  MoveL 10079 to (-40.2, 152.67, 144.49) mm, rotated rx -180 ry 0 rz 180 deg; joints [-142.671, 73.983, -86.26, 142.029, 80.265, 7.518]
  Call Extruder(400.11411)
  MoveL 10080 to (-40.24, 152.44, 144.49) mm, rotated rx -180 ry 0 rz 180 deg; joints [-142.718, 73.976, -86.267, 142.076, 80.248, 7.518]
  MoveL 10081 to (-40.24, 152.44, 144.49) mm, rotated rx -180 ry 0 rz 180 deg; joints [-142.718, 73.976, -86.267, 142.076, 80.248, 7.518]
  Call Extruder(400.25109)
  MoveL 10082 to (-40.29, 152.2, 144.49) mm, rotated rx 180 ry 0 rz -180 deg; joints [-142.77, 73.969, -86.275, 142.127, 80.23, 7.518]
  MoveL 10083 to (-40.29, 152.2, 144.49) mm, rotated rx 180 ry 0 rz -180 deg; joints [-142.77, 73.969, -86.275, 142.127, 80.23, 7.518]
  Call Extruder(400.38745)
  MoveL 10084 to (-40.34, 151.95, 144.49) mm, rotated rx 180 ry 0 rz -180 deg; joints [-142.822, 73.961, -86.282, 142.177, 80.211, 7.519]
  MoveL 10085 to (-40.34, 151.95, 144.49) mm, rotated rx 180 ry 0 rz -180 deg; joints [-142.822, 73.961, -86.282, 142.177, 80.211, 7.519]
  Call Extruder(400.52321)
  MoveL 10086 to (-40.39, 151.7, 144.49) mm, rotated rx -180 ry 0 rz -180 deg; joints [-142.874, 73.954, -86.29, 142.228, 80.193, 7.519]
  MoveL 10087 to (-40.39, 151.7, 144.49) mm, rotated rx -180 ry 0 rz -180 deg; joints [-142.874, 73.954, -86.29, 142.228, 80.193, 7.519]
  Call Extruder(400.65835)
  MoveL 10088 to (-40.44, 151.45, 144.49) mm, rotated rx -180 ry 0 rz 180 deg; joints [-142.926, 73.947, -86.297, 142.279, 80.174, 7.519]
  MoveL 10089 to (-40.44, 151.45, 144.49) mm, rotated rx -180 ry 0 rz 180 deg; joints [-142.926, 73.947, -86.297, 142.279, 80.174, 7.519]
  Call Extruder(400.79289)
  MoveL 10090 to (-40.49, 151.2, 144.49) mm, rotated rx -180 ry 0 rz 180 deg; joints [-142.978, 73.939, -86.304, 142.33, 80.156, 7.52]
  MoveL 10091 to (-40.49, 151.2, 144.49) mm, rotated rx -180 ry 0 rz 180 deg; joints [-142.978, 73.939, -86.304, 142.33, 80.156, 7.52]
  Call Extruder(400.92681)
  MoveL 10092 to (-40.54, 150.95, 144.49) mm, rotated rx -180 ry 0 rz -180 deg; joints [-143.031, 73.932, -86.312, 142.381, 80.137, 7.52]
  MoveL 10093 to (-40.54, 150.95, 144.49) mm, rotated rx -180 ry 0 rz -180 deg; joints [-143.031, 73.932, -86.312, 142.381, 80.137, 7.52]
  Call Extruder(401.07467)
  MoveL 10094 to (-40.59, 150.67, 144.49) mm, rotated rx -180 ry 0 rz 180 deg; joints [-143.088, 73.923, -86.321, 142.437, 80.116, 7.521]
  MoveL 10095 to (-40.59, 150.67, 144.49) mm, rotated rx -180 ry 0 rz 180 deg; joints [-143.088, 73.923, -86.321, 142.437, 80.116, 7.521]
  Call Extruder(401.23639)
  MoveL 10096 to (-40.64, 150.37, 144.49) mm, rotated rx 180 ry 0 rz 180 deg; joints [-143.15, 73.914, -86.33, 142.498, 80.092, 7.522]
  MoveL 10097 to (-40.64, 150.37, 144.49) mm, rotated rx 180 ry 0 rz 180 deg; joints [-143.15, 73.914, -86.33, 142.498, 80.092, 7.522]
  Call Extruder(401.39739)
  MoveL 10098 to (-40.69, 150.06, 144.49) mm, rotated rx -180 ry 0 rz 180 deg; joints [-143.213, 73.904, -86.34, 142.558, 80.069, 7.523]
  MoveL 10099 to (-40.69, 150.06, 144.49) mm, rotated rx -180 ry 0 rz 180 deg; joints [-143.213, 73.904, -86.34, 142.558, 80.069, 7.523]
  Call Extruder(401.55766)
  MoveL 10100 to (-40.74, 149.76, 144.49) mm, rotated rx 180 ry 0 rz 180 deg; joints [-143.276, 73.894, -86.35, 142.619, 80.045, 7.524]
  MoveL 10101 to (-40.74, 149.76, 144.49) mm, rotated rx 180 ry 0 rz 180 deg; joints [-143.276, 73.894, -86.35, 142.619, 80.045, 7.524]
  Call Extruder(401.71721)
  MoveL 10102 to (-40.78, 149.45, 144.49) mm, rotated rx 180 ry 0 rz 180 deg; joints [-143.338, 73.885, -86.359, 142.681, 80.022, 7.525]
  MoveL 10103 to (-40.78, 149.45, 144.49) mm, rotated rx 180 ry 0 rz 180 deg; joints [-143.338, 73.885, -86.359, 142.681, 80.022, 7.525]
  Call Extruder(401.87602)
  MoveL 10104 to (-40.83, 149.14, 144.49) mm, rotated rx -180 ry 0 rz -180 deg; joints [-143.401, 73.875, -86.369, 142.742, 79.998, 7.526]
  MoveL 10105 to (-40.83, 149.14, 144.49) mm, rotated rx -180 ry 0 rz -180 deg; joints [-143.401, 73.875, -86.369, 142.742, 79.998, 7.526]
  Call Extruder(402.05468)
  MoveL 10106 to (-40.88, 148.8, 144.49) mm, rotated rx 180 ry 0 rz 180 deg; joints [-143.471, 73.864, -86.38, 142.81, 79.971, 7.527]
  MoveL 10107 to (-40.88, 148.8, 144.49) mm, rotated rx 180 ry 0 rz 180 deg; joints [-143.471, 73.864, -86.38, 142.81, 79.971, 7.527]
  Call Extruder(402.25313)
  MoveL 10108 to (-40.93, 148.41, 144.49) mm, rotated rx -180 ry 0 rz 180 deg; joints [-143.549, 73.851, -86.393, 142.885, 79.94, 7.53]
  MoveL 10109 to (-40.93, 148.41, 144.49) mm, rotated rx -180 ry 0 rz 180 deg; joints [-143.549, 73.851, -86.393, 142.885, 79.94, 7.53]
  Call Extruder(402.45070)
  MoveL 10110 to (-40.97, 148.02, 144.49) mm, rotated rx 180 ry 0 rz -180 deg; joints [-143.627, 73.838, -86.406, 142.961, 79.909, 7.532]
  MoveL 10111 to (-40.97, 148.02, 144.49) mm, rotated rx 180 ry 0 rz -180 deg; joints [-143.627, 73.838, -86.406, 142.961, 79.909, 7.532]
  Call Extruder(402.64741)
  MoveL 10112 to (-41.02, 147.63, 144.49) mm, rotated rx -180 ry 0 rz 180 deg; joints [-143.705, 73.825, -86.419, 143.037, 79.878, 7.534]
  MoveL 10113 to (-41.02, 147.63, 144.49) mm, rotated rx -180 ry 0 rz 180 deg; joints [-143.705, 73.825, -86.419, 143.037, 79.878, 7.534]
  Call Extruder(402.84324)
  MoveL 10114 to (-41.06, 147.25, 144.49) mm, rotated rx -180 ry 0 rz 180 deg; joints [-143.783, 73.812, -86.432, 143.112, 79.847, 7.536]
  MoveL 10115 to (-41.06, 147.25, 144.49) mm, rotated rx -180 ry 0 rz 180 deg; joints [-143.783, 73.812, -86.432, 143.112, 79.847, 7.536]
  Call Extruder(403.13864)
  MoveL 10116 to (-41.11, 146.66, 144.49) mm, rotated rx 180 ry 0 rz -180 deg; joints [-143.899, 73.791, -86.453, 143.225, 79.799, 7.541]
  MoveL 10117 to (-41.11, 146.66, 144.49) mm, rotated rx 180 ry 0 rz -180 deg; joints [-143.899, 73.791, -86.453, 143.225, 79.799, 7.541]
  Call Extruder(403.43270)
  MoveL 10118 to (-41.16, 146.07, 144.49) mm, rotated rx 180 ry 0 rz 180 deg; joints [-144.015, 73.77, -86.473, 143.337, 79.75, 7.545]
  MoveL 10119 to (-41.16, 146.07, 144.49) mm, rotated rx 180 ry 0 rz 180 deg; joints [-144.015, 73.77, -86.473, 143.337, 79.75, 7.545]
  Call Extruder(403.72544)
  MoveL 10120 to (-41.2, 145.48, 144.49) mm, rotated rx -180 ry 0 rz 180 deg; joints [-144.131, 73.749, -86.494, 143.45, 79.702, 7.549]
  MoveL 10121 to (-41.2, 145.48, 144.49) mm, rotated rx -180 ry 0 rz 180 deg; joints [-144.131, 73.749, -86.494, 143.45, 79.702, 7.549]
  Call Extruder(404.29889)
  MoveL 10122 to (-41.25, 144.32, 144.49) mm, rotated rx 180 ry 0 rz 180 deg; joints [-144.355, 73.705, -86.536, 143.666, 79.603, 7.561]
  MoveL 10123 to (-41.25, 144.32, 144.49) mm, rotated rx 180 ry 0 rz 180 deg; joints [-144.355, 73.705, -86.536, 143.666, 79.603, 7.561]
  Call Extruder(405.01285)
  MoveL 10124 to (-41.29, 142.86, 144.49) mm, rotated rx 180 ry 0 rz -180 deg; joints [-144.635, 73.65, -86.59, 143.937, 79.478, 7.575]
  Call Extruder(447.07768)
  MoveL 10125 to (-41.29, 57.14, 144.49) mm, rotated rx 180 ry 0 rz -180 deg; joints [-164.153, 70.836, -88.802, 163.384, 72.739, 5.06]
  Call Extruder(447.50624)
  MoveL 10126 to (-41.27, 56.26, 144.49) mm, rotated rx -180 ry 0 rz -180 deg; joints [-164.382, 70.815, -88.815, 163.62, 72.687, 4.999]
  MoveL 10127 to (-41.27, 56.26, 144.49) mm, rotated rx -180 ry 0 rz -180 deg; joints [-164.382, 70.815, -88.815, 163.62, 72.687, 4.999]
  Call Extruder(448.07969)
  MoveL 10128 to (-41.23, 55.1, 144.49) mm, rotated rx -180 ry 0 rz 180 deg; joints [-164.686, 70.787, -88.833, 163.934, 72.615, 4.918]
  MoveL 10129 to (-41.23, 55.1, 144.49) mm, rotated rx -180 ry 0 rz 180 deg; joints [-164.686, 70.787, -88.833, 163.934, 72.615, 4.918]
  Call Extruder(448.51400)
  MoveL 10130 to (-41.18, 54.23, 144.49) mm, rotated rx -180 ry 0 rz 180 deg; joints [-164.915, 70.764, -88.847, 164.17, 72.561, 4.857]
  MoveL 10131 to (-41.18, 54.23, 144.49) mm, rotated rx -180 ry 0 rz 180 deg; joints [-164.915, 70.764, -88.847, 164.17, 72.561, 4.857]
  Call Extruder(448.80807)
  MoveL 10132 to (-41.13, 53.64, 144.49) mm, rotated rx 180 ry 0 rz -180 deg; joints [-165.068, 70.748, -88.857, 164.328, 72.522, 4.817]
  MoveL 10133 to (-41.13, 53.64, 144.49) mm, rotated rx 180 ry 0 rz -180 deg; joints [-165.068, 70.748, -88.857, 164.328, 72.522, 4.817]
  Call Extruder(449.10346)
  MoveL 10134 to (-41.09, 53.05, 144.49) mm, rotated rx -180 ry 0 rz 180 deg; joints [-165.222, 70.732, -88.867, 164.486, 72.484, 4.776]
  MoveL 10135 to (-41.09, 53.05, 144.49) mm, rotated rx -180 ry 0 rz 180 deg; joints [-165.222, 70.732, -88.867, 164.486, 72.484, 4.776]
  Call Extruder(449.34970)
  MoveL 10136 to (-41.04, 52.56, 144.49) mm, rotated rx -180 ry 0 rz -180 deg; joints [-165.349, 70.718, -88.876, 164.616, 72.452, 4.742]
  MoveL 10137 to (-41.04, 52.56, 144.49) mm, rotated rx -180 ry 0 rz -180 deg; joints [-165.349, 70.718, -88.876, 164.616, 72.452, 4.742]
  Call Extruder(449.54640)
  MoveL 10138 to (-40.99, 52.17, 144.49) mm, rotated rx 180 ry 0 rz 180 deg; joints [-165.449, 70.707, -88.883, 164.72, 72.426, 4.716]
  MoveL 10139 to (-40.99, 52.17, 144.49) mm, rotated rx 180 ry 0 rz 180 deg; joints [-165.449, 70.707, -88.883, 164.72, 72.426, 4.716]
  Call Extruder(449.74398)
  MoveL 10140 to (-40.95, 51.78, 144.49) mm, rotated rx -180 ry 0 rz -180 deg; joints [-165.549, 70.695, -88.891, 164.823, 72.399, 4.689]
  MoveL 10141 to (-40.95, 51.78, 144.49) mm, rotated rx -180 ry 0 rz -180 deg; joints [-165.549, 70.695, -88.891, 164.823, 72.399, 4.689]
  Call Extruder(449.94242)
  MoveL 10142 to (-40.9, 51.4, 144.49) mm, rotated rx 180 ry 0 rz -180 deg; joints [-165.65, 70.684, -88.898, 164.927, 72.373, 4.662]
  MoveL 10143 to (-40.9, 51.4, 144.49) mm, rotated rx 180 ry 0 rz -180 deg; joints [-165.65, 70.684, -88.898, 164.927, 72.373, 4.662]
  Call Extruder(450.14173)
  MoveL 10144 to (-40.86, 51.01, 144.49) mm, rotated rx -180 ry 0 rz -180 deg; joints [-165.751, 70.672, -88.905, 165.03, 72.347, 4.636]
  MoveL 10145 to (-40.86, 51.01, 144.49) mm, rotated rx -180 ry 0 rz -180 deg; joints [-165.751, 70.672, -88.905, 165.03, 72.347, 4.636]
  Call Extruder(450.30055)
  MoveL 10146 to (-40.81, 50.7, 144.49) mm, rotated rx 180 ry 0 rz -180 deg; joints [-165.829, 70.662, -88.911, 165.111, 72.325, 4.615]
  MoveL 10147 to (-40.81, 50.7, 144.49) mm, rotated rx 180 ry 0 rz -180 deg; joints [-165.829, 70.662, -88.911, 165.111, 72.325, 4.615]
  Call Extruder(450.46009)
  MoveL 10148 to (-40.76, 50.4, 144.49) mm, rotated rx 180 ry 0 rz -180 deg; joints [-165.908, 70.652, -88.917, 165.193, 72.303, 4.594]
  MoveL 10149 to (-40.76, 50.4, 144.49) mm, rotated rx 180 ry 0 rz -180 deg; joints [-165.908, 70.652, -88.917, 165.193, 72.303, 4.594]
  Call Extruder(450.62036)
  MoveL 10150 to (-40.71, 50.09, 144.49) mm, rotated rx -180 ry 0 rz -180 deg; joints [-165.987, 70.642, -88.924, 165.274, 72.281, 4.574]
  MoveL 10151 to (-40.71, 50.09, 144.49) mm, rotated rx -180 ry 0 rz -180 deg; joints [-165.987, 70.642, -88.924, 165.274, 72.281, 4.574]
  Call Extruder(450.78136)
  MoveL 10152 to (-40.66, 49.79, 144.49) mm, rotated rx 180 ry 0 rz -180 deg; joints [-166.066, 70.632, -88.93, 165.355, 72.259, 4.553]
  MoveL 10153 to (-40.66, 49.79, 144.49) mm, rotated rx 180 ry 0 rz -180 deg; joints [-166.066, 70.632, -88.93, 165.355, 72.259, 4.553]
  Call Extruder(450.94309)
  MoveL 10154 to (-40.61, 49.48, 144.49) mm, rotated rx 180 ry 0 rz 180 deg; joints [-166.145, 70.623, -88.936, 165.436, 72.238, 4.532]
  MoveL 10155 to (-40.61, 49.48, 144.49) mm, rotated rx 180 ry 0 rz 180 deg; joints [-166.145, 70.623, -88.936, 165.436, 72.238, 4.532]
  Call Extruder(451.10554)
  MoveL 10156 to (-40.57, 49.17, 144.49) mm, rotated rx -180 ry 0 rz -180 deg; joints [-166.224, 70.613, -88.942, 165.518, 72.216, 4.511]
  MoveL 10157 to (-40.57, 49.17, 144.49) mm, rotated rx -180 ry 0 rz -180 deg; joints [-166.224, 70.613, -88.942, 165.518, 72.216, 4.511]
  Call Extruder(451.23946)
  MoveL 10158 to (-40.52, 48.93, 144.49) mm, rotated rx 180 ry 0 rz -180 deg; joints [-166.288, 70.604, -88.947, 165.584, 72.197, 4.494]
  MoveL 10159 to (-40.52, 48.93, 144.49) mm, rotated rx 180 ry 0 rz -180 deg; joints [-166.288, 70.604, -88.947, 165.584, 72.197, 4.494]
  Call Extruder(451.37400)
  MoveL 10160 to (-40.47, 48.68, 144.49) mm, rotated rx 180 ry 0 rz 180 deg; joints [-166.352, 70.595, -88.953, 165.65, 72.178, 4.477]
  MoveL 10161 to (-40.47, 48.68, 144.49) mm, rotated rx 180 ry 0 rz 180 deg; joints [-166.352, 70.595, -88.953, 165.65, 72.178, 4.477]
  Call Extruder(451.50914)
  MoveL 10162 to (-40.42, 48.43, 144.49) mm, rotated rx 180 ry 0 rz 180 deg; joints [-166.416, 70.586, -88.958, 165.715, 72.159, 4.46]
  MoveL 10163 to (-40.42, 48.43, 144.49) mm, rotated rx 180 ry 0 rz 180 deg; joints [-166.416, 70.586, -88.958, 165.715, 72.159, 4.46]
  Call Extruder(451.64490)
  MoveL 10164 to (-40.37, 48.18, 144.49) mm, rotated rx -180 ry 0 rz 180 deg; joints [-166.48, 70.577, -88.964, 165.781, 72.141, 4.443]
  MoveL 10165 to (-40.37, 48.18, 144.49) mm, rotated rx -180 ry 0 rz 180 deg; joints [-166.48, 70.577, -88.964, 165.781, 72.141, 4.443]
  Call Extruder(451.78127)
  MoveL 10166 to (-40.32, 47.93, 144.49) mm, rotated rx 180 ry 0 rz 180 deg; joints [-166.544, 70.569, -88.969, 165.847, 72.122, 4.426]
  MoveL 10167 to (-40.32, 47.93, 144.49) mm, rotated rx 180 ry 0 rz 180 deg; joints [-166.544, 70.569, -88.969, 165.847, 72.122, 4.426]
  Call Extruder(451.91824)
  MoveL 10168 to (-40.27, 47.68, 144.49) mm, rotated rx 180 ry 0 rz 180 deg; joints [-166.608, 70.56, -88.974, 165.914, 72.104, 4.409]
  MoveL 10169 to (-40.27, 47.68, 144.49) mm, rotated rx 180 ry 0 rz 180 deg; joints [-166.608, 70.56, -88.974, 165.914, 72.104, 4.409]
  Call Extruder(452.05583)
  MoveL 10170 to (-40.22, 47.43, 144.49) mm, rotated rx -180 ry 0 rz 180 deg; joints [-166.673, 70.551, -88.98, 165.98, 72.085, 4.392]
  MoveL 10171 to (-40.22, 47.43, 144.49) mm, rotated rx -180 ry 0 rz 180 deg; joints [-166.673, 70.551, -88.98, 165.98, 72.085, 4.392]
  Call Extruder(452.16955)
  MoveL 10172 to (-40.17, 47.23, 144.49) mm, rotated rx -180 ry 0 rz -180 deg; joints [-166.725, 70.544, -88.984, 166.034, 72.069, 4.378]
  MoveL 10173 to (-40.17, 47.23, 144.49) mm, rotated rx -180 ry 0 rz -180 deg; joints [-166.725, 70.544, -88.984, 166.034, 72.069, 4.378]
  Call Extruder(452.28373)
  MoveL 10174 to (-40.13, 47.02, 144.49) mm, rotated rx 180 ry 0 rz 180 deg; joints [-166.778, 70.536, -88.989, 166.088, 72.054, 4.364]
  MoveL 10175 to (-40.13, 47.02, 144.49) mm, rotated rx 180 ry 0 rz 180 deg; joints [-166.778, 70.536, -88.989, 166.088, 72.054, 4.364]
  Call Extruder(452.39837)
  MoveL 10176 to (-40.08, 46.82, 144.49) mm, rotated rx 180 ry 0 rz -180 deg; joints [-166.83, 70.529, -88.993, 166.142, 72.038, 4.35]
  MoveL 10177 to (-40.08, 46.82, 144.49) mm, rotated rx 180 ry 0 rz -180 deg; joints [-166.83, 70.529, -88.993, 166.142, 72.038, 4.35]
  Call Extruder(452.51345)
  MoveL 10178 to (-40.04, 46.61, 144.49) mm, rotated rx -180 ry 0 rz -180 deg; joints [-166.883, 70.522, -88.998, 166.197, 72.022, 4.336]
  MoveL 10179 to (-40.04, 46.61, 144.49) mm, rotated rx -180 ry 0 rz -180 deg; joints [-166.883, 70.522, -88.998, 166.197, 72.022, 4.336]
  Call Extruder(452.63569)
  MoveL 10180 to (-39.98, 46.4, 144.49) mm, rotated rx -180 ry 0 rz -180 deg; joints [-166.937, 70.513, -89.003, 166.253, 72.005, 4.322]
  MoveL 10181 to (-39.98, 46.4, 144.49) mm, rotated rx -180 ry 0 rz -180 deg; joints [-166.937, 70.513, -89.003, 166.253, 72.005, 4.322]
  Call Extruder(452.76536)
  MoveL 10182 to (-39.92, 46.18, 144.49) mm, rotated rx -180 ry 0 rz 180 deg; joints [-166.994, 70.503, -89.009, 166.311, 71.986, 4.308]
  MoveL 10183 to (-39.92, 46.18, 144.49) mm, rotated rx -180 ry 0 rz 180 deg; joints [-166.994, 70.503, -89.009, 166.311, 71.986, 4.308]
  Call Extruder(452.89558)
  MoveL 10184 to (-39.85, 45.95, 144.49) mm, rotated rx 180 ry 0 rz -180 deg; joints [-167.051, 70.494, -89.015, 166.369, 71.966, 4.293]
  MoveL 10185 to (-39.85, 45.95, 144.49) mm, rotated rx 180 ry 0 rz -180 deg; joints [-167.051, 70.494, -89.015, 166.369, 71.966, 4.293]
  Call Extruder(453.02638)
  MoveL 10186 to (-39.78, 45.73, 144.49) mm, rotated rx 180 ry 0 rz -180 deg; joints [-167.107, 70.484, -89.021, 166.427, 71.947, 4.279]
  MoveL 10187 to (-39.78, 45.73, 144.49) mm, rotated rx 180 ry 0 rz -180 deg; joints [-167.107, 70.484, -89.021, 166.427, 71.947, 4.279]
  Call Extruder(453.15773)
  MoveL 10188 to (-39.71, 45.5, 144.49) mm, rotated rx 180 ry 0 rz 180 deg; joints [-167.164, 70.475, -89.026, 166.486, 71.928, 4.264]
  MoveL 10189 to (-39.71, 45.5, 144.49) mm, rotated rx 180 ry 0 rz 180 deg; joints [-167.164, 70.475, -89.026, 166.486, 71.928, 4.264]
  Call Extruder(453.26964)
  MoveL 10190 to (-39.65, 45.32, 144.49) mm, rotated rx 180 ry 0 rz 180 deg; joints [-167.212, 70.466, -89.031, 166.535, 71.911, 4.252]
  MoveL 10191 to (-39.65, 45.32, 144.49) mm, rotated rx 180 ry 0 rz 180 deg; joints [-167.212, 70.466, -89.031, 166.535, 71.911, 4.252]
  Call Extruder(453.38198)
  MoveL 10192 to (-39.59, 45.13, 144.49) mm, rotated rx -180 ry 0 rz 180 deg; joints [-167.26, 70.458, -89.037, 166.584, 71.895, 4.239]
  MoveL 10193 to (-39.59, 45.13, 144.49) mm, rotated rx -180 ry 0 rz 180 deg; joints [-167.26, 70.458, -89.037, 166.584, 71.895, 4.239]
  Call Extruder(453.49477)
  MoveL 10194 to (-39.53, 44.94, 144.49) mm, rotated rx -180 ry 0 rz -180 deg; joints [-167.307, 70.449, -89.042, 166.633, 71.878, 4.227]
  MoveL 10195 to (-39.53, 44.94, 144.49) mm, rotated rx -180 ry 0 rz -180 deg; joints [-167.307, 70.449, -89.042, 166.633, 71.878, 4.227]
  Call Extruder(453.60801)
  MoveL 10196 to (-39.47, 44.75, 144.49) mm, rotated rx 180 ry 0 rz 180 deg; joints [-167.355, 70.441, -89.047, 166.682, 71.862, 4.215]
  MoveL 10197 to (-39.47, 44.75, 144.49) mm, rotated rx 180 ry 0 rz 180 deg; joints [-167.355, 70.441, -89.047, 166.682, 71.862, 4.215]
  Call Extruder(453.72169)
  MoveL 10198 to (-39.41, 44.56, 144.49) mm, rotated rx -180 ry 0 rz -180 deg; joints [-167.403, 70.433, -89.052, 166.731, 71.845, 4.202]
  MoveL 10199 to (-39.41, 44.56, 144.49) mm, rotated rx -180 ry 0 rz -180 deg; joints [-167.403, 70.433, -89.052, 166.731, 71.845, 4.202]
  Call Extruder(453.90365)
  MoveL 10200 to (-39.29, 44.27, 144.49) mm, rotated rx 180 ry 0 rz 180 deg; joints [-167.475, 70.418, -89.061, 166.805, 71.816, 4.185]
  MoveL 10201 to (-39.29, 44.27, 144.49) mm, rotated rx 180 ry 0 rz 180 deg; joints [-167.475, 70.418, -89.061, 166.805, 71.816, 4.185]
  Call Extruder(454.08636)
  MoveL 10202 to (-39.16, 43.98, 144.49) mm, rotated rx -180 ry 0 rz 180 deg; joints [-167.548, 70.403, -89.07, 166.88, 71.788, 4.166]
  MoveL 10203 to (-39.16, 43.98, 144.49) mm, rotated rx -180 ry 0 rz 180 deg; joints [-167.548, 70.403, -89.07, 166.88, 71.788, 4.166]
  Call Extruder(454.25678)
  MoveL 10204 to (-39.05, 43.71, 144.49) mm, rotated rx -180 ry 0 rz -180 deg; joints [-167.615, 70.389, -89.078, 166.949, 71.761, 4.15]
  MoveL 10205 to (-39.05, 43.71, 144.49) mm, rotated rx -180 ry 0 rz -180 deg; joints [-167.615, 70.389, -89.078, 166.949, 71.761, 4.15]
  Call Extruder(454.41476)
  MoveL 10206 to (-38.94, 43.46, 144.49) mm, rotated rx -180 ry 0 rz 180 deg; joints [-167.677, 70.375, -89.086, 167.012, 71.736, 4.134]
  MoveL 10207 to (-38.94, 43.46, 144.49) mm, rotated rx -180 ry 0 rz 180 deg; joints [-167.677, 70.375, -89.086, 167.012, 71.736, 4.134]
  Call Extruder(454.57335)
  MoveL 10208 to (-38.84, 43.21, 144.49) mm, rotated rx 180 ry 0 rz -180 deg; joints [-167.739, 70.362, -89.094, 167.076, 71.711, 4.119]
  MoveL 10209 to (-38.84, 43.21, 144.49) mm, rotated rx 180 ry 0 rz -180 deg; joints [-167.739, 70.362, -89.094, 167.076, 71.711, 4.119]
  Call Extruder(454.77952)
  MoveL 10210 to (-38.66, 42.91, 144.49) mm, rotated rx -180 ry 0 rz -180 deg; joints [-167.813, 70.343, -89.106, 167.151, 71.675, 4.102]
  MoveL 10211 to (-38.66, 42.91, 144.49) mm, rotated rx -180 ry 0 rz -180 deg; joints [-167.813, 70.343, -89.106, 167.151, 71.675, 4.102]
  Call Extruder(454.98646)
  MoveL 10212 to (-38.49, 42.6, 144.49) mm, rotated rx -180 ry 0 rz -180 deg; joints [-167.886, 70.323, -89.117, 167.226, 71.639, 4.085]
  MoveL 10213 to (-38.49, 42.6, 144.49) mm, rotated rx -180 ry 0 rz -180 deg; joints [-167.886, 70.323, -89.117, 167.226, 71.639, 4.085]
  Call Extruder(455.19419)
  MoveL 10214 to (-38.31, 42.3, 144.49) mm, rotated rx -180 ry 0 rz -180 deg; joints [-167.96, 70.304, -89.129, 167.301, 71.604, 4.068]
  MoveL 10215 to (-38.31, 42.3, 144.49) mm, rotated rx -180 ry 0 rz -180 deg; joints [-167.96, 70.304, -89.129, 167.301, 71.604, 4.068]
  Call Extruder(455.40269)
  MoveL 10216 to (-38.14, 41.99, 144.49) mm, rotated rx -180 ry 0 rz -180 deg; joints [-168.033, 70.284, -89.141, 167.376, 71.568, 4.051]
  MoveL 10217 to (-38.14, 41.99, 144.49) mm, rotated rx -180 ry 0 rz -180 deg; joints [-168.033, 70.284, -89.141, 167.376, 71.568, 4.051]
  Call Extruder(455.58224)
  MoveL 10218 to (-37.96, 41.75, 144.49) mm, rotated rx -180 ry 0 rz 180 deg; joints [-168.091, 70.265, -89.151, 167.434, 71.535, 4.038]
  MoveL 10219 to (-37.96, 41.75, 144.49) mm, rotated rx -180 ry 0 rz 180 deg; joints [-168.091, 70.265, -89.151, 167.434, 71.535, 4.038]
  Call Extruder(455.91567)
  MoveL 10220 to (-37.63, 41.3, 144.49) mm, rotated rx -180 ry 0 rz 180 deg; joints [-168.197, 70.231, -89.172, 167.542, 71.474, 4.015]
  MoveL 10221 to (-37.63, 41.3, 144.49) mm, rotated rx -180 ry 0 rz 180 deg; joints [-168.197, 70.231, -89.172, 167.542, 71.474, 4.015]
  Call Extruder(456.25030)
  MoveL 10222 to (-37.3, 40.85, 144.49) mm, rotated rx 180 ry 0 rz 180 deg; joints [-168.304, 70.196, -89.192, 167.65, 71.413, 3.992]
  Call Extruder(457.07823)
  MoveL 10223 to (-36.39, 39.81, 144.49) mm, rotated rx 180 ry 0 rz 180 deg; joints [-168.541, 70.104, -89.246, 167.89, 71.254, 3.945]
  Call Extruder(457.90614)
  MoveL 10224 to (-35.35, 38.9, 144.49) mm, rotated rx 180 ry 0 rz 180 deg; joints [-168.739, 70.003, -89.303, 168.087, 71.085, 3.912]
  Call Extruder(458.07344)
  MoveL 10225 to (-35.13, 38.73, 144.49) mm, rotated rx 180 ry 0 rz 180 deg; joints [-168.773, 69.981, -89.316, 168.12, 71.05, 3.908]
  MoveL 10226 to (-35.13, 38.73, 144.49) mm, rotated rx 180 ry 0 rz 180 deg; joints [-168.773, 69.981, -89.316, 168.12, 71.05, 3.908]
  Call Extruder(458.40687)
  MoveL 10227 to (-34.68, 38.4, 144.49) mm, rotated rx -180 ry 0 rz 180 deg; joints [-168.84, 69.938, -89.34, 168.187, 70.98, 3.899]
  MoveL 10228 to (-34.68, 38.4, 144.49) mm, rotated rx -180 ry 0 rz 180 deg; joints [-168.84, 69.938, -89.34, 168.187, 70.98, 3.899]
  Call Extruder(458.73911)
  MoveL 10229 to (-34.23, 38.08, 144.49) mm, rotated rx 180 ry 0 rz 180 deg; joints [-168.908, 69.895, -89.364, 168.254, 70.909, 3.89]
  MoveL 10230 to (-34.23, 38.08, 144.49) mm, rotated rx 180 ry 0 rz 180 deg; joints [-168.908, 69.895, -89.364, 168.254, 70.909, 3.89]
  Call Extruder(458.85681)
  MoveL 10231 to (-34.05, 37.98, 144.49) mm, rotated rx 180 ry 0 rz 180 deg; joints [-168.927, 69.879, -89.373, 168.272, 70.884, 3.889]
  MoveL 10232 to (-34.05, 37.98, 144.49) mm, rotated rx 180 ry 0 rz 180 deg; joints [-168.927, 69.879, -89.373, 168.272, 70.884, 3.889]
  Call Extruder(459.06453)
  MoveL 10233 to (-33.75, 37.8, 144.49) mm, rotated rx 180 ry 0 rz 180 deg; joints [-168.96, 69.851, -89.388, 168.304, 70.838, 3.887]
  MoveL 10234 to (-33.75, 37.8, 144.49) mm, rotated rx 180 ry 0 rz 180 deg; joints [-168.96, 69.851, -89.388, 168.304, 70.838, 3.887]
  Call Extruder(459.27147)
  MoveL 10235 to (-33.45, 37.63, 144.49) mm, rotated rx -180 ry 0 rz 180 deg; joints [-168.993, 69.823, -89.404, 168.336, 70.793, 3.885]
  MoveL 10236 to (-33.45, 37.63, 144.49) mm, rotated rx -180 ry 0 rz 180 deg; joints [-168.993, 69.823, -89.404, 168.336, 70.793, 3.885]
  Call Extruder(459.47764)
  MoveL 10237 to (-33.14, 37.45, 144.49) mm, rotated rx -180 ry 0 rz -180 deg; joints [-169.026, 69.794, -89.42, 168.367, 70.748, 3.883]
  MoveL 10238 to (-33.14, 37.45, 144.49) mm, rotated rx -180 ry 0 rz -180 deg; joints [-169.026, 69.794, -89.42, 168.367, 70.748, 3.883]
  Call Extruder(459.65932)
  MoveL 10239 to (-32.87, 37.31, 144.49) mm, rotated rx -180 ry 0 rz 180 deg; joints [-169.052, 69.769, -89.434, 168.391, 70.707, 3.883]
  MoveL 10240 to (-32.87, 37.31, 144.49) mm, rotated rx -180 ry 0 rz 180 deg; joints [-169.052, 69.769, -89.434, 168.391, 70.707, 3.883]
  Call Extruder(459.81731)
  MoveL 10241 to (-32.62, 37.2, 144.49) mm, rotated rx -180 ry 0 rz 180 deg; joints [-169.068, 69.746, -89.446, 168.407, 70.672, 3.884]
  MoveL 10242 to (-32.62, 37.2, 144.49) mm, rotated rx -180 ry 0 rz 180 deg; joints [-169.068, 69.746, -89.446, 168.407, 70.672, 3.884]
  Call Extruder(459.97470)
  MoveL 10243 to (-32.37, 37.09, 144.49) mm, rotated rx -180 ry 0 rz -180 deg; joints [-169.085, 69.724, -89.459, 168.422, 70.636, 3.886]
  MoveL 10244 to (-32.37, 37.09, 144.49) mm, rotated rx -180 ry 0 rz -180 deg; joints [-169.085, 69.724, -89.459, 168.422, 70.636, 3.886]
  Call Extruder(460.13371)
  MoveL 10245 to (-32.11, 36.99, 144.49) mm, rotated rx -180 ry 0 rz 180 deg; joints [-169.101, 69.701, -89.471, 168.437, 70.6, 3.888]
  MoveL 10246 to (-32.11, 36.99, 144.49) mm, rotated rx -180 ry 0 rz 180 deg; joints [-169.101, 69.701, -89.471, 168.437, 70.6, 3.888]
  Call Extruder(460.28213)
  MoveL 10247 to (-31.88, 36.89, 144.49) mm, rotated rx 180 ry 0 rz 180 deg; joints [-169.116, 69.679, -89.483, 168.45, 70.567, 3.89]
  MoveL 10248 to (-31.88, 36.89, 144.49) mm, rotated rx 180 ry 0 rz 180 deg; joints [-169.116, 69.679, -89.483, 168.45, 70.567, 3.89]
  Call Extruder(460.43006)
  MoveL 10249 to (-31.64, 36.79, 144.49) mm, rotated rx -180 ry 0 rz -180 deg; joints [-169.132, 69.657, -89.495, 168.464, 70.533, 3.891]
  MoveL 10250 to (-31.64, 36.79, 144.49) mm, rotated rx -180 ry 0 rz -180 deg; joints [-169.132, 69.657, -89.495, 168.464, 70.533, 3.891]
  Call Extruder(460.54351)
  MoveL 10251 to (-31.45, 36.73, 144.49) mm, rotated rx -180 ry 0 rz 180 deg; joints [-169.139, 69.64, -89.504, 168.47, 70.507, 3.894]
  MoveL 10252 to (-31.45, 36.73, 144.49) mm, rotated rx -180 ry 0 rz 180 deg; joints [-169.139, 69.64, -89.504, 168.47, 70.507, 3.894]
  Call Extruder(460.65653)
  MoveL 10253 to (-31.26, 36.67, 144.49) mm, rotated rx -180 ry 0 rz -180 deg; joints [-169.146, 69.623, -89.513, 168.476, 70.481, 3.897]
  MoveL 10254 to (-31.26, 36.67, 144.49) mm, rotated rx -180 ry 0 rz -180 deg; joints [-169.146, 69.623, -89.513, 168.476, 70.481, 3.897]
  Call Extruder(460.76910)
  MoveL 10255 to (-31.07, 36.61, 144.49) mm, rotated rx -180 ry 0 rz -180 deg; joints [-169.154, 69.607, -89.522, 168.482, 70.455, 3.9]
  MoveL 10256 to (-31.07, 36.61, 144.49) mm, rotated rx -180 ry 0 rz -180 deg; joints [-169.154, 69.607, -89.522, 168.482, 70.455, 3.9]
  Call Extruder(460.88122)
  MoveL 10257 to (-30.88, 36.55, 144.49) mm, rotated rx 180 ry 0 rz 180 deg; joints [-169.161, 69.59, -89.531, 168.487, 70.429, 3.903]
  MoveL 10258 to (-30.88, 36.55, 144.49) mm, rotated rx 180 ry 0 rz 180 deg; joints [-169.161, 69.59, -89.531, 168.487, 70.429, 3.903]
  Call Extruder(460.99290)
  MoveL 10259 to (-30.7, 36.49, 144.49) mm, rotated rx 180 ry 0 rz 180 deg; joints [-169.168, 69.573, -89.54, 168.493, 70.403, 3.906]
  MoveL 10260 to (-30.7, 36.49, 144.49) mm, rotated rx 180 ry 0 rz 180 deg; joints [-169.168, 69.573, -89.54, 168.493, 70.403, 3.906]
  Call Extruder(461.12397)
  MoveL 10261 to (-30.47, 36.42, 144.49) mm, rotated rx -180 ry 0 rz -180 deg; joints [-169.175, 69.553, -89.551, 168.499, 70.372, 3.91]
  MoveL 10262 to (-30.47, 36.42, 144.49) mm, rotated rx -180 ry 0 rz -180 deg; joints [-169.175, 69.553, -89.551, 168.499, 70.372, 3.91]
  Call Extruder(461.25448)
  MoveL 10263 to (-30.25, 36.35, 144.49) mm, rotated rx 180 ry 0 rz -180 deg; joints [-169.182, 69.532, -89.562, 168.504, 70.342, 3.914]
  MoveL 10264 to (-30.25, 36.35, 144.49) mm, rotated rx 180 ry 0 rz -180 deg; joints [-169.182, 69.532, -89.562, 168.504, 70.342, 3.914]
  Call Extruder(461.38443)
  MoveL 10265 to (-30.02, 36.28, 144.49) mm, rotated rx -180 ry 0 rz -180 deg; joints [-169.19, 69.512, -89.572, 168.51, 70.311, 3.918]
  MoveL 10266 to (-30.02, 36.28, 144.49) mm, rotated rx -180 ry 0 rz -180 deg; joints [-169.19, 69.512, -89.572, 168.51, 70.311, 3.918]
  Call Extruder(461.51381)
  MoveL 10267 to (-29.8, 36.22, 144.49) mm, rotated rx -180 ry 0 rz -180 deg; joints [-169.197, 69.492, -89.583, 168.515, 70.28, 3.922]
  MoveL 10268 to (-29.8, 36.22, 144.49) mm, rotated rx -180 ry 0 rz -180 deg; joints [-169.197, 69.492, -89.583, 168.515, 70.28, 3.922]
  Call Extruder(461.63577)
  MoveL 10269 to (-29.59, 36.16, 144.49) mm, rotated rx -180 ry 0 rz 180 deg; joints [-169.202, 69.473, -89.593, 168.518, 70.251, 3.926]
  MoveL 10270 to (-29.59, 36.16, 144.49) mm, rotated rx -180 ry 0 rz 180 deg; joints [-169.202, 69.473, -89.593, 168.518, 70.251, 3.926]
  Call Extruder(461.75062)
  MoveL 10271 to (-29.38, 36.12, 144.49) mm, rotated rx -180 ry 0 rz -180 deg; joints [-169.203, 69.455, -89.603, 168.517, 70.224, 3.932]
  MoveL 10272 to (-29.38, 36.12, 144.49) mm, rotated rx -180 ry 0 rz -180 deg; joints [-169.203, 69.455, -89.603, 168.517, 70.224, 3.932]
  Call Extruder(461.86501)
  MoveL 10273 to (-29.18, 36.07, 144.49) mm, rotated rx -180 ry 0 rz -180 deg; joints [-169.205, 69.437, -89.612, 168.517, 70.197, 3.937]
  MoveL 10274 to (-29.18, 36.07, 144.49) mm, rotated rx -180 ry 0 rz -180 deg; joints [-169.205, 69.437, -89.612, 168.517, 70.197, 3.937]
  Call Extruder(461.97895)
  MoveL 10275 to (-28.97, 36.03, 144.49) mm, rotated rx 180 ry 0 rz -180 deg; joints [-169.207, 69.419, -89.622, 168.517, 70.17, 3.942]
  MoveL 10276 to (-28.97, 36.03, 144.49) mm, rotated rx 180 ry 0 rz -180 deg; joints [-169.207, 69.419, -89.622, 168.517, 70.17, 3.942]
  Call Extruder(462.09244)
  MoveL 10277 to (-28.77, 35.98, 144.49) mm, rotated rx -180 ry 0 rz 180 deg; joints [-169.208, 69.401, -89.631, 168.517, 70.143, 3.947]
  MoveL 10278 to (-28.77, 35.98, 144.49) mm, rotated rx -180 ry 0 rz 180 deg; joints [-169.208, 69.401, -89.631, 168.517, 70.143, 3.947]
  Call Extruder(462.22973)
  MoveL 10279 to (-28.52, 35.93, 144.49) mm, rotated rx 180 ry 0 rz 180 deg; joints [-169.209, 69.379, -89.643, 168.515, 70.11, 3.954]
  MoveL 10280 to (-28.52, 35.93, 144.49) mm, rotated rx 180 ry 0 rz 180 deg; joints [-169.209, 69.379, -89.643, 168.515, 70.11, 3.954]
  Call Extruder(462.36640)
  MoveL 10281 to (-28.27, 35.88, 144.49) mm, rotated rx -180 ry 0 rz -180 deg; joints [-169.209, 69.356, -89.654, 168.513, 70.077, 3.961]
  MoveL 10282 to (-28.27, 35.88, 144.49) mm, rotated rx -180 ry 0 rz -180 deg; joints [-169.209, 69.356, -89.654, 168.513, 70.077, 3.961]
  Call Extruder(462.50246)
  MoveL 10283 to (-28.02, 35.83, 144.49) mm, rotated rx 180 ry 0 rz -180 deg; joints [-169.21, 69.334, -89.666, 168.512, 70.044, 3.968]
  MoveL 10284 to (-28.02, 35.83, 144.49) mm, rotated rx 180 ry 0 rz -180 deg; joints [-169.21, 69.334, -89.666, 168.512, 70.044, 3.968]
  Call Extruder(462.63791)
  MoveL 10285 to (-27.77, 35.78, 144.49) mm, rotated rx 180 ry 0 rz 180 deg; joints [-169.21, 69.312, -89.677, 168.51, 70.011, 3.975]
  MoveL 10286 to (-27.77, 35.78, 144.49) mm, rotated rx 180 ry 0 rz 180 deg; joints [-169.21, 69.312, -89.677, 168.51, 70.011, 3.975]
  Call Extruder(462.77275)
  MoveL 10287 to (-27.52, 35.73, 144.49) mm, rotated rx 180 ry 0 rz 180 deg; joints [-169.211, 69.29, -89.688, 168.508, 69.978, 3.982]
  MoveL 10288 to (-27.52, 35.73, 144.49) mm, rotated rx 180 ry 0 rz 180 deg; joints [-169.211, 69.29, -89.688, 168.508, 69.978, 3.982]
  Call Extruder(462.90698)
  MoveL 10289 to (-27.27, 35.68, 144.49) mm, rotated rx 180 ry 0 rz -180 deg; joints [-169.212, 69.268, -89.7, 168.506, 69.945, 3.989]
  MoveL 10290 to (-27.27, 35.68, 144.49) mm, rotated rx 180 ry 0 rz -180 deg; joints [-169.212, 69.268, -89.7, 168.506, 69.945, 3.989]
  Call Extruder(463.04061)
  MoveL 10291 to (-27.03, 35.63, 144.49) mm, rotated rx 180 ry 0 rz -180 deg; joints [-169.212, 69.246, -89.711, 168.504, 69.912, 3.996]
  MoveL 10292 to (-27.03, 35.63, 144.49) mm, rotated rx 180 ry 0 rz -180 deg; joints [-169.212, 69.246, -89.711, 168.504, 69.912, 3.996]
  Call Extruder(463.20270)
  MoveL 10293 to (-26.72, 35.59, 144.49) mm, rotated rx -180 ry 0 rz 180 deg; joints [-169.21, 69.219, -89.725, 168.499, 69.872, 4.005]
  MoveL 10294 to (-26.72, 35.59, 144.49) mm, rotated rx -180 ry 0 rz 180 deg; joints [-169.21, 69.219, -89.725, 168.499, 69.872, 4.005]
  Call Extruder(463.36408)
  MoveL 10295 to (-26.41, 35.54, 144.49) mm, rotated rx 180 ry 0 rz 180 deg; joints [-169.207, 69.191, -89.739, 168.492, 69.832, 4.015]
  MoveL 10296 to (-26.41, 35.54, 144.49) mm, rotated rx 180 ry 0 rz 180 deg; joints [-169.207, 69.191, -89.739, 168.492, 69.832, 4.015]
  Call Extruder(463.52472)
  MoveL 10297 to (-26.11, 35.49, 144.49) mm, rotated rx 180 ry 0 rz 180 deg; joints [-169.204, 69.164, -89.752, 168.486, 69.792, 4.025]
  MoveL 10298 to (-26.11, 35.49, 144.49) mm, rotated rx 180 ry 0 rz 180 deg; joints [-169.204, 69.164, -89.752, 168.486, 69.792, 4.025]
  Call Extruder(463.68463)
  MoveL 10299 to (-25.8, 35.44, 144.49) mm, rotated rx -180 ry 0 rz 180 deg; joints [-169.201, 69.137, -89.766, 168.48, 69.753, 4.035]
  MoveL 10300 to (-25.8, 35.44, 144.49) mm, rotated rx -180 ry 0 rz 180 deg; joints [-169.201, 69.137, -89.766, 168.48, 69.753, 4.035]
  Call Extruder(463.84382)
  MoveL 10301 to (-25.5, 35.39, 144.49) mm, rotated rx 180 ry 0 rz -180 deg; joints [-169.198, 69.11, -89.78, 168.474, 69.713, 4.044]
  MoveL 10302 to (-25.5, 35.39, 144.49) mm, rotated rx 180 ry 0 rz -180 deg; joints [-169.198, 69.11, -89.78, 168.474, 69.713, 4.044]
  Call Extruder(464.00228)
  MoveL 10303 to (-25.19, 35.34, 144.49) mm, rotated rx -180 ry 0 rz 180 deg; joints [-169.195, 69.083, -89.793, 168.468, 69.673, 4.054]
  MoveL 10304 to (-25.19, 35.34, 144.49) mm, rotated rx -180 ry 0 rz 180 deg; joints [-169.195, 69.083, -89.793, 168.468, 69.673, 4.054]
  Call Extruder(464.20116)
  MoveL 10305 to (-24.8, 35.3, 144.49) mm, rotated rx -180 ry 0 rz -180 deg; joints [-169.187, 69.048, -89.81, 168.455, 69.623, 4.068]
  MoveL 10306 to (-24.8, 35.3, 144.49) mm, rotated rx -180 ry 0 rz -180 deg; joints [-169.187, 69.048, -89.81, 168.455, 69.623, 4.068]
  Call Extruder(464.39916)
  MoveL 10307 to (-24.42, 35.25, 144.49) mm, rotated rx 180 ry 0 rz 180 deg; joints [-169.178, 69.014, -89.827, 168.442, 69.573, 4.082]
  MoveL 10308 to (-24.42, 35.25, 144.49) mm, rotated rx 180 ry 0 rz 180 deg; joints [-169.178, 69.014, -89.827, 168.442, 69.573, 4.082]
  Call Extruder(464.59630)
  MoveL 10309 to (-24.03, 35.21, 144.49) mm, rotated rx -180 ry 0 rz 180 deg; joints [-169.17, 68.98, -89.844, 168.43, 69.524, 4.096]
  MoveL 10310 to (-24.03, 35.21, 144.49) mm, rotated rx -180 ry 0 rz 180 deg; joints [-169.17, 68.98, -89.844, 168.43, 69.524, 4.096]
  Call Extruder(464.79258)
  MoveL 10311 to (-23.64, 35.16, 144.49) mm, rotated rx 180 ry 0 rz 180 deg; joints [-169.161, 68.945, -89.861, 168.417, 69.474, 4.111]
  MoveL 10312 to (-23.64, 35.16, 144.49) mm, rotated rx 180 ry 0 rz 180 deg; joints [-169.161, 68.945, -89.861, 168.417, 69.474, 4.111]
  Call Extruder(465.03826)
  MoveL 10313 to (-23.15, 35.11, 144.49) mm, rotated rx -180 ry 0 rz 180 deg; joints [-169.147, 68.902, -89.882, 168.397, 69.412, 4.13]
  MoveL 10314 to (-23.15, 35.11, 144.49) mm, rotated rx -180 ry 0 rz 180 deg; joints [-169.147, 68.902, -89.882, 168.397, 69.412, 4.13]
  Call Extruder(465.33299)
  MoveL 10315 to (-22.56, 35.07, 144.49) mm, rotated rx -180 ry 0 rz -180 deg; joints [-169.127, 68.85, -89.908, 168.369, 69.338, 4.154]
  MoveL 10316 to (-22.56, 35.07, 144.49) mm, rotated rx -180 ry 0 rz -180 deg; joints [-169.127, 68.85, -89.908, 168.369, 69.338, 4.154]
  Call Extruder(465.62639)
  MoveL 10317 to (-21.97, 35.02, 144.49) mm, rotated rx 180 ry 0 rz 180 deg; joints [-169.107, 68.797, -89.933, 168.342, 69.263, 4.178]
  MoveL 10318 to (-21.97, 35.02, 144.49) mm, rotated rx 180 ry 0 rz 180 deg; joints [-169.107, 68.797, -89.933, 168.342, 69.263, 4.178]
  Call Extruder(466.05972)
  MoveL 10319 to (-21.1, 34.97, 144.49) mm, rotated rx -180 ry 0 rz -180 deg; joints [-169.069, 68.72, -89.97, 168.293, 69.154, 4.217]
  MoveL 10320 to (-21.1, 34.97, 144.49) mm, rotated rx -180 ry 0 rz -180 deg; joints [-169.069, 68.72, -89.97, 168.293, 69.154, 4.217]
  Call Extruder(466.63188)
  MoveL 10321 to (-19.94, 34.93, 144.49) mm, rotated rx -180 ry 0 rz -180 deg; joints [-169.014, 68.617, -90.018, 168.222, 69.009, 4.271]
  MoveL 10322 to (-19.94, 34.93, 144.49) mm, rotated rx -180 ry 0 rz -180 deg; joints [-169.014, 68.617, -90.018, 168.222, 69.009, 4.271]
  Call Extruder(467.05971)
  MoveL 10323 to (-19.06, 34.91, 144.49) mm, rotated rx 180 ry 0 rz 180 deg; joints [-168.967, 68.539, -90.055, 168.164, 68.902, 4.314]
  Call Extruder(583.70842)
  MoveL 10324 to (219.06, 34.91, 144.49) mm, rotated rx -180 ry 0 rz 160 deg; joints [-52.528, 61.546, -92.021, 74.822, 98.759, 29.306]
  MoveL 10325 to (219.06, 34.91, 144.49) mm, rotated rx -180 ry 0 rz 160 deg; joints [-52.528, 61.546, -92.021, 74.822, 98.759, 29.306]
  Call Extruder(584.42399)
  MoveL 10326 to (220.52, 34.95, 144.49) mm, rotated rx -180 ry 0 rz 160 deg; joints [-51.959, 61.648, -92.007, 74.302, 99.005, 29.115]
  MoveL 10327 to (220.52, 34.95, 144.49) mm, rotated rx -180 ry 0 rz 160 deg; joints [-51.959, 61.648, -92.007, 74.302, 99.005, 29.115]
  Call Extruder(584.99873)
  MoveL 10328 to (221.68, 35, 144.49) mm, rotated rx 180 ry 0 rz 160 deg; joints [-51.515, 61.731, -91.995, 73.895, 99.195, 28.961]
  MoveL 10329 to (221.68, 35, 144.49) mm, rotated rx 180 ry 0 rz 160 deg; joints [-51.515, 61.731, -91.995, 73.895, 99.195, 28.961]
  Call Extruder(585.29212)
  MoveL 10330 to (222.27, 35.05, 144.49) mm, rotated rx 180 ry 0 rz 160 deg; joints [-51.3, 61.776, -91.989, 73.696, 99.285, 28.88]
  MoveL 10331 to (222.27, 35.05, 144.49) mm, rotated rx 180 ry 0 rz 160 deg; joints [-51.3, 61.776, -91.989, 73.696, 99.285, 28.88]
  Call Extruder(585.58685)
  MoveL 10332 to (222.86, 35.09, 144.49) mm, rotated rx -180 ry 0 rz 160 deg; joints [-51.086, 61.82, -91.983, 73.498, 99.373, 28.8]
  MoveL 10333 to (222.86, 35.09, 144.49) mm, rotated rx -180 ry 0 rz 160 deg; joints [-51.086, 61.82, -91.983, 73.498, 99.373, 28.8]
  Call Extruder(585.88292)
  MoveL 10334 to (223.45, 35.14, 144.49) mm, rotated rx 180 ry 0 rz 160 deg; joints [-50.874, 61.865, -91.976, 73.301, 99.461, 28.719]
  MoveL 10335 to (223.45, 35.14, 144.49) mm, rotated rx 180 ry 0 rz 160 deg; joints [-50.874, 61.865, -91.976, 73.301, 99.461, 28.719]
  Call Extruder(586.07919)
  MoveL 10336 to (223.83, 35.18, 144.49) mm, rotated rx -180 ry 0 rz 160 deg; joints [-50.739, 61.896, -91.972, 73.176, 99.515, 28.666]
  MoveL 10337 to (223.83, 35.18, 144.49) mm, rotated rx -180 ry 0 rz 160 deg; joints [-50.739, 61.896, -91.972, 73.176, 99.515, 28.666]
  Call Extruder(586.27633)
  MoveL 10338 to (224.22, 35.23, 144.49) mm, rotated rx 180 ry 0 rz 160 deg; joints [-50.606, 61.927, -91.967, 73.051, 99.569, 28.611]
  MoveL 10339 to (224.22, 35.23, 144.49) mm, rotated rx 180 ry 0 rz 160 deg; joints [-50.606, 61.927, -91.967, 73.051, 99.569, 28.611]
  Call Extruder(586.47434)
  MoveL 10340 to (224.61, 35.28, 144.49) mm, rotated rx 180 ry 0 rz 160 deg; joints [-50.473, 61.957, -91.962, 72.928, 99.622, 28.557]
  MoveL 10341 to (224.61, 35.28, 144.49) mm, rotated rx 180 ry 0 rz 160 deg; joints [-50.473, 61.957, -91.962, 72.928, 99.622, 28.557]
  Call Extruder(586.67322)
  MoveL 10342 to (225, 35.32, 144.49) mm, rotated rx -180 ry 0 rz 160 deg; joints [-50.341, 61.988, -91.958, 72.804, 99.675, 28.503]
  MoveL 10343 to (225, 35.32, 144.49) mm, rotated rx -180 ry 0 rz 160 deg; joints [-50.341, 61.988, -91.958, 72.804, 99.675, 28.503]
  Call Extruder(586.85230)
  MoveL 10344 to (225.34, 35.37, 144.49) mm, rotated rx 180 ry 0 rz 160 deg; joints [-50.226, 62.017, -91.954, 72.696, 99.72, 28.454]
  MoveL 10345 to (225.34, 35.37, 144.49) mm, rotated rx 180 ry 0 rz 160 deg; joints [-50.226, 62.017, -91.954, 72.696, 99.72, 28.454]
  Call Extruder(587.01148)
  MoveL 10346 to (225.65, 35.42, 144.49) mm, rotated rx -180 ry 0 rz 160 deg; joints [-50.126, 62.042, -91.95, 72.602, 99.759, 28.411]
  MoveL 10347 to (225.65, 35.42, 144.49) mm, rotated rx -180 ry 0 rz 160 deg; joints [-50.126, 62.042, -91.95, 72.602, 99.759, 28.411]
  Call Extruder(587.17139)
  MoveL 10348 to (225.96, 35.47, 144.49) mm, rotated rx 180 ry 0 rz 160 deg; joints [-50.027, 62.068, -91.946, 72.509, 99.797, 28.367]
  MoveL 10349 to (225.96, 35.47, 144.49) mm, rotated rx 180 ry 0 rz 160 deg; joints [-50.027, 62.068, -91.946, 72.509, 99.797, 28.367]
  Call Extruder(587.33203)
  MoveL 10350 to (226.26, 35.51, 144.49) mm, rotated rx -180 ry 0 rz 160 deg; joints [-49.928, 62.093, -91.942, 72.416, 99.835, 28.324]
  MoveL 10351 to (226.26, 35.51, 144.49) mm, rotated rx -180 ry 0 rz 160 deg; joints [-49.928, 62.093, -91.942, 72.416, 99.835, 28.324]
  Call Extruder(587.49340)
  MoveL 10352 to (226.57, 35.56, 144.49) mm, rotated rx 180 ry 0 rz 160 deg; joints [-49.83, 62.119, -91.938, 72.323, 99.873, 28.28]
  MoveL 10353 to (226.57, 35.56, 144.49) mm, rotated rx 180 ry 0 rz 160 deg; joints [-49.83, 62.119, -91.938, 72.323, 99.873, 28.28]
  Call Extruder(587.65549)
  MoveL 10354 to (226.87, 35.61, 144.49) mm, rotated rx 180 ry 0 rz 160 deg; joints [-49.732, 62.144, -91.934, 72.231, 99.91, 28.237]
  MoveL 10355 to (226.87, 35.61, 144.49) mm, rotated rx 180 ry 0 rz 160 deg; joints [-49.732, 62.144, -91.934, 72.231, 99.91, 28.237]
  Call Extruder(587.80369)
  MoveL 10356 to (227.15, 35.66, 144.49) mm, rotated rx 180 ry 0 rz 160 deg; joints [-49.645, 62.168, -91.93, 72.148, 99.943, 28.197]
  MoveL 10357 to (227.15, 35.66, 144.49) mm, rotated rx 180 ry 0 rz 160 deg; joints [-49.645, 62.168, -91.93, 72.148, 99.943, 28.197]
  Call Extruder(587.93792)
  MoveL 10358 to (227.4, 35.71, 144.49) mm, rotated rx 180 ry 0 rz 160 deg; joints [-49.569, 62.19, -91.927, 72.076, 99.971, 28.161]
  MoveL 10359 to (227.4, 35.71, 144.49) mm, rotated rx 180 ry 0 rz 160 deg; joints [-49.569, 62.19, -91.927, 72.076, 99.971, 28.161]
  Call Extruder(588.07276)
  MoveL 10360 to (227.65, 35.76, 144.49) mm, rotated rx 180 ry 0 rz 160 deg; joints [-49.493, 62.211, -91.924, 72.004, 99.999, 28.125]
  MoveL 10361 to (227.65, 35.76, 144.49) mm, rotated rx 180 ry 0 rz 160 deg; joints [-49.493, 62.211, -91.924, 72.004, 99.999, 28.125]
  Call Extruder(588.20822)
  MoveL 10362 to (227.9, 35.81, 144.49) mm, rotated rx -180 ry 0 rz 160 deg; joints [-49.418, 62.233, -91.92, 71.932, 100.027, 28.089]
  MoveL 10363 to (227.9, 35.81, 144.49) mm, rotated rx -180 ry 0 rz 160 deg; joints [-49.418, 62.233, -91.92, 71.932, 100.027, 28.089]
  Call Extruder(588.34428)
  MoveL 10364 to (228.15, 35.86, 144.49) mm, rotated rx -180 ry 0 rz 160 deg; joints [-49.343, 62.255, -91.917, 71.86, 100.054, 28.053]
  MoveL 10365 to (228.15, 35.86, 144.49) mm, rotated rx -180 ry 0 rz 160 deg; joints [-49.343, 62.255, -91.917, 71.86, 100.054, 28.053]
  Call Extruder(588.48095)
  MoveL 10366 to (228.4, 35.91, 144.49) mm, rotated rx 180 ry 0 rz 160 deg; joints [-49.267, 62.277, -91.913, 71.788, 100.082, 28.016]
  MoveL 10367 to (228.4, 35.91, 144.49) mm, rotated rx 180 ry 0 rz 160 deg; joints [-49.267, 62.277, -91.913, 71.788, 100.082, 28.016]
  Call Extruder(588.61823)
  MoveL 10368 to (228.65, 35.96, 144.49) mm, rotated rx 180 ry 0 rz 160 deg; joints [-49.192, 62.299, -91.91, 71.717, 100.109, 27.98]
  MoveL 10369 to (228.65, 35.96, 144.49) mm, rotated rx 180 ry 0 rz 160 deg; joints [-49.192, 62.299, -91.91, 71.717, 100.109, 27.98]
  Call Extruder(588.74391)
  MoveL 10370 to (228.87, 36, 144.49) mm, rotated rx -180 ry 0 rz 160 deg; joints [-49.125, 62.318, -91.906, 71.653, 100.133, 27.947]
  MoveL 10371 to (228.87, 36, 144.49) mm, rotated rx -180 ry 0 rz 160 deg; joints [-49.125, 62.318, -91.906, 71.653, 100.133, 27.947]
  Call Extruder(588.85785)
  MoveL 10372 to (229.08, 36.05, 144.49) mm, rotated rx 180 ry 0 rz 160 deg; joints [-49.065, 62.337, -91.904, 71.596, 100.155, 27.917]
  MoveL 10373 to (229.08, 36.05, 144.49) mm, rotated rx 180 ry 0 rz 160 deg; joints [-49.065, 62.337, -91.904, 71.596, 100.155, 27.917]
  Call Extruder(588.97225)
  MoveL 10374 to (229.28, 36.09, 144.49) mm, rotated rx 180 ry 0 rz 160 deg; joints [-49.006, 62.355, -91.901, 71.539, 100.176, 27.888]
  MoveL 10375 to (229.28, 36.09, 144.49) mm, rotated rx 180 ry 0 rz 160 deg; joints [-49.006, 62.355, -91.901, 71.539, 100.176, 27.888]
  Call Extruder(589.08710)
  MoveL 10376 to (229.48, 36.14, 144.49) mm, rotated rx 180 ry 0 rz 160 deg; joints [-48.947, 62.373, -91.898, 71.482, 100.197, 27.858]
  MoveL 10377 to (229.48, 36.14, 144.49) mm, rotated rx 180 ry 0 rz 160 deg; joints [-48.947, 62.373, -91.898, 71.482, 100.197, 27.858]
  Call Extruder(589.20240)
  MoveL 10378 to (229.69, 36.18, 144.49) mm, rotated rx 180 ry 0 rz 160 deg; joints [-48.888, 62.391, -91.895, 71.425, 100.218, 27.828]
  MoveL 10379 to (229.69, 36.18, 144.49) mm, rotated rx 180 ry 0 rz 160 deg; joints [-48.888, 62.391, -91.895, 71.425, 100.218, 27.828]
  Call Extruder(589.26695)
  MoveL 10380 to (229.8, 36.22, 144.49) mm, rotated rx -180 ry 0 rz 160 deg; joints [-48.858, 62.402, -91.893, 71.396, 100.228, 27.811]
  MoveL 10381 to (229.8, 36.22, 144.49) mm, rotated rx -180 ry 0 rz 160 deg; joints [-48.858, 62.402, -91.893, 71.396, 100.228, 27.811]
  Call Extruder(589.39662)
  MoveL 10382 to (230.02, 36.28, 144.49) mm, rotated rx 180 ry 0 rz 160 deg; joints [-48.799, 62.424, -91.889, 71.339, 100.247, 27.778]
  MoveL 10383 to (230.02, 36.28, 144.49) mm, rotated rx 180 ry 0 rz 160 deg; joints [-48.799, 62.424, -91.889, 71.339, 100.247, 27.778]
  Call Extruder(589.52685)
  MoveL 10384 to (230.25, 36.35, 144.49) mm, rotated rx -180 ry 0 rz 160 deg; joints [-48.741, 62.445, -91.886, 71.283, 100.266, 27.744]
  MoveL 10385 to (230.25, 36.35, 144.49) mm, rotated rx -180 ry 0 rz 160 deg; joints [-48.741, 62.445, -91.886, 71.283, 100.266, 27.744]
  Call Extruder(589.65764)
  MoveL 10386 to (230.47, 36.42, 144.49) mm, rotated rx -180 ry 0 rz 160 deg; joints [-48.682, 62.467, -91.882, 71.226, 100.285, 27.711]
  MoveL 10387 to (230.47, 36.42, 144.49) mm, rotated rx -180 ry 0 rz 160 deg; joints [-48.682, 62.467, -91.882, 71.226, 100.285, 27.711]
  Call Extruder(589.78900)
  MoveL 10388 to (230.7, 36.49, 144.49) mm, rotated rx 180 ry 0 rz 160 deg; joints [-48.624, 62.488, -91.879, 71.169, 100.304, 27.677]
  MoveL 10389 to (230.7, 36.49, 144.49) mm, rotated rx 180 ry 0 rz 160 deg; joints [-48.624, 62.488, -91.879, 71.169, 100.304, 27.677]
  Call Extruder(589.90090)
  MoveL 10390 to (230.88, 36.55, 144.49) mm, rotated rx 180 ry 0 rz 160 deg; joints [-48.577, 62.507, -91.875, 71.123, 100.319, 27.649]
  MoveL 10391 to (230.88, 36.55, 144.49) mm, rotated rx 180 ry 0 rz 160 deg; joints [-48.577, 62.507, -91.875, 71.123, 100.319, 27.649]
  Call Extruder(590.01324)
  MoveL 10392 to (231.07, 36.61, 144.49) mm, rotated rx -180 ry 0 rz 160 deg; joints [-48.529, 62.525, -91.872, 71.076, 100.334, 27.62]
  MoveL 10393 to (231.07, 36.61, 144.49) mm, rotated rx -180 ry 0 rz 160 deg; joints [-48.529, 62.525, -91.872, 71.076, 100.334, 27.62]
  Call Extruder(590.12603)
  MoveL 10394 to (231.26, 36.67, 144.49) mm, rotated rx 180 ry 0 rz 160 deg; joints [-48.482, 62.544, -91.869, 71.03, 100.349, 27.592]
  MoveL 10395 to (231.26, 36.67, 144.49) mm, rotated rx 180 ry 0 rz 160 deg; joints [-48.482, 62.544, -91.869, 71.03, 100.349, 27.592]
  Call Extruder(590.23926)
  MoveL 10396 to (231.45, 36.73, 144.49) mm, rotated rx 180 ry 0 rz 160 deg; joints [-48.435, 62.562, -91.866, 70.984, 100.364, 27.564]
  MoveL 10397 to (231.45, 36.73, 144.49) mm, rotated rx 180 ry 0 rz 160 deg; joints [-48.435, 62.562, -91.866, 70.984, 100.364, 27.564]
  Call Extruder(590.35294)
  MoveL 10398 to (231.64, 36.79, 144.49) mm, rotated rx -180 ry 0 rz 160 deg; joints [-48.388, 62.58, -91.863, 70.938, 100.379, 27.535]
  MoveL 10399 to (231.64, 36.79, 144.49) mm, rotated rx -180 ry 0 rz 160 deg; joints [-48.388, 62.58, -91.863, 70.938, 100.379, 27.535]
  Call Extruder(590.53490)
  MoveL 10400 to (231.93, 36.91, 144.49) mm, rotated rx 180 ry 0 rz 160 deg; joints [-48.324, 62.611, -91.858, 70.873, 100.397, 27.49]
  MoveL 10401 to (231.93, 36.91, 144.49) mm, rotated rx 180 ry 0 rz 160 deg; joints [-48.324, 62.611, -91.858, 70.873, 100.397, 27.49]
  Call Extruder(590.71761)
  MoveL 10402 to (232.22, 37.03, 144.49) mm, rotated rx -180 ry 0 rz 160 deg; joints [-48.259, 62.642, -91.852, 70.809, 100.414, 27.445]
  MoveL 10403 to (232.22, 37.03, 144.49) mm, rotated rx -180 ry 0 rz 160 deg; joints [-48.259, 62.642, -91.852, 70.809, 100.414, 27.445]
  Call Extruder(590.88803)
  MoveL 10404 to (232.49, 37.15, 144.49) mm, rotated rx 180 ry 0 rz 160 deg; joints [-48.201, 62.67, -91.847, 70.751, 100.43, 27.403]
  MoveL 10405 to (232.49, 37.15, 144.49) mm, rotated rx 180 ry 0 rz 160 deg; joints [-48.201, 62.67, -91.847, 70.751, 100.43, 27.403]
  Call Extruder(591.04603)
  MoveL 10406 to (232.74, 37.26, 144.49) mm, rotated rx 180 ry 0 rz 160 deg; joints [-48.148, 62.697, -91.843, 70.697, 100.444, 27.365]
  MoveL 10407 to (232.74, 37.26, 144.49) mm, rotated rx 180 ry 0 rz 160 deg; joints [-48.148, 62.697, -91.843, 70.697, 100.444, 27.365]
  Call Extruder(591.20464)
  MoveL 10408 to (232.99, 37.36, 144.49) mm, rotated rx 180 ry 0 rz 160 deg; joints [-48.095, 62.723, -91.838, 70.644, 100.458, 27.326]
  MoveL 10409 to (232.99, 37.36, 144.49) mm, rotated rx 180 ry 0 rz 160 deg; joints [-48.095, 62.723, -91.838, 70.644, 100.458, 27.326]
  Call Extruder(591.41080)
  MoveL 10410 to (233.29, 37.54, 144.49) mm, rotated rx 180 ry 0 rz 160 deg; joints [-48.044, 62.759, -91.832, 70.591, 100.467, 27.277]
  MoveL 10411 to (233.29, 37.54, 144.49) mm, rotated rx 180 ry 0 rz 160 deg; joints [-48.044, 62.759, -91.832, 70.591, 100.467, 27.277]
  Call Extruder(591.61775)
  MoveL 10412 to (233.6, 37.71, 144.49) mm, rotated rx -180 ry 0 rz 160 deg; joints [-47.994, 62.795, -91.825, 70.538, 100.476, 27.228]
  MoveL 10413 to (233.6, 37.71, 144.49) mm, rotated rx -180 ry 0 rz 160 deg; joints [-47.994, 62.795, -91.825, 70.538, 100.476, 27.228]
  Call Extruder(591.82547)
  MoveL 10414 to (233.9, 37.89, 144.49) mm, rotated rx 180 ry 0 rz 180 deg; joints [-27.144, 58.124, -92.29, 31.783, 119.982, 17.205]
  MoveL 10415 to (233.9, 37.89, 144.49) mm, rotated rx 180 ry 0 rz 180 deg; joints [-27.144, 58.124, -92.29, 31.783, 119.982, 17.205]
  Call Extruder(592.03398)
  MoveL 10416 to (234.21, 38.07, 144.49) mm, rotated rx 180 ry 0 rz 180 deg; joints [-27.156, 58.166, -92.288, 31.784, 119.942, 17.186]
  MoveL 10417 to (234.21, 38.07, 144.49) mm, rotated rx 180 ry 0 rz 180 deg; joints [-27.156, 58.166, -92.288, 31.784, 119.942, 17.186]
  Call Extruder(592.21352)
  MoveL 10418 to (234.45, 38.24, 144.49) mm, rotated rx -180 ry 0 rz -180 deg; joints [-27.187, 58.201, -92.287, 31.807, 119.902, 17.181]
  MoveL 10419 to (234.45, 38.24, 144.49) mm, rotated rx -180 ry 0 rz -180 deg; joints [-27.187, 58.201, -92.287, 31.807, 119.902, 17.181]
  Call Extruder(592.54693)
  MoveL 10420 to (234.9, 38.57, 144.49) mm, rotated rx 180 ry 0 rz 180 deg; joints [-27.245, 58.266, -92.285, 31.851, 119.828, 17.172]
  MoveL 10421 to (234.9, 38.57, 144.49) mm, rotated rx 180 ry 0 rz 180 deg; joints [-27.245, 58.266, -92.285, 31.851, 119.828, 17.172]
  Call Extruder(592.88153)
  MoveL 10422 to (235.35, 38.9, 144.49) mm, rotated rx -180 ry 0 rz 180 deg; joints [-27.302, 58.331, -92.283, 31.894, 119.755, 17.162]
  Call Extruder(593.70948)
  MoveL 10423 to (236.39, 39.81, 144.49) mm, rotated rx 180 ry 0 rz 180 deg; joints [-27.525, 58.489, -92.278, 32.089, 119.55, 17.184]
  Call Extruder(594.53743)
  MoveL 10424 to (237.3, 40.85, 144.49) mm, rotated rx -180 ry 0 rz 180 deg; joints [-27.851, 58.64, -92.272, 32.4, 119.321, 17.264]
  Call Extruder(594.70473)
  MoveL 10425 to (237.47, 41.07, 144.49) mm, rotated rx 180 ry 0 rz 180 deg; joints [-27.932, 58.669, -92.271, 32.479, 119.271, 17.288]
  MoveL 10426 to (237.47, 41.07, 144.49) mm, rotated rx 180 ry 0 rz 180 deg; joints [-27.932, 58.669, -92.271, 32.479, 119.271, 17.288]
  Call Extruder(595.03814)
  MoveL 10427 to (237.8, 41.52, 144.49) mm, rotated rx 180 ry 0 rz -180 deg; joints [-28.091, 58.728, -92.268, 32.634, 119.172, 17.335]
  MoveL 10428 to (237.8, 41.52, 144.49) mm, rotated rx 180 ry 0 rz -180 deg; joints [-28.091, 58.728, -92.268, 32.634, 119.172, 17.335]
  Call Extruder(595.37037)
  MoveL 10429 to (238.12, 41.98, 144.49) mm, rotated rx 180 ry 0 rz 180 deg; joints [-28.249, 58.787, -92.266, 32.788, 119.074, 17.381]
  MoveL 10430 to (238.12, 41.98, 144.49) mm, rotated rx 180 ry 0 rz 180 deg; joints [-28.249, 58.787, -92.266, 32.788, 119.074, 17.381]
  Call Extruder(595.48807)
  MoveL 10431 to (238.22, 42.15, 144.49) mm, rotated rx -180 ry 0 rz 180 deg; joints [-28.315, 58.806, -92.265, 32.855, 119.036, 17.404]
  MoveL 10432 to (238.22, 42.15, 144.49) mm, rotated rx -180 ry 0 rz 180 deg; joints [-28.315, 58.806, -92.265, 32.855, 119.036, 17.404]
  Call Extruder(595.69580)
  MoveL 10433 to (238.4, 42.45, 144.49) mm, rotated rx -180 ry 0 rz 180 deg; joints [-28.434, 58.841, -92.263, 32.973, 118.97, 17.444]
  MoveL 10434 to (238.4, 42.45, 144.49) mm, rotated rx -180 ry 0 rz 180 deg; joints [-28.434, 58.841, -92.263, 32.973, 118.97, 17.444]
  Call Extruder(595.90274)
  MoveL 10435 to (238.57, 42.75, 144.49) mm, rotated rx 180 ry 0 rz 180 deg; joints [-28.552, 58.876, -92.261, 33.09, 118.904, 17.483]
  MoveL 10436 to (238.57, 42.75, 144.49) mm, rotated rx 180 ry 0 rz 180 deg; joints [-28.552, 58.876, -92.261, 33.09, 118.904, 17.483]
  Call Extruder(596.10891)
  MoveL 10437 to (238.75, 43.06, 144.49) mm, rotated rx 180 ry 0 rz 180 deg; joints [-28.669, 58.911, -92.26, 33.207, 118.838, 17.522]
  MoveL 10438 to (238.75, 43.06, 144.49) mm, rotated rx 180 ry 0 rz 180 deg; joints [-28.669, 58.911, -92.26, 33.207, 118.838, 17.522]
  Call Extruder(596.29060)
  MoveL 10439 to (238.89, 43.33, 144.49) mm, rotated rx 180 ry 0 rz 180 deg; joints [-28.78, 58.941, -92.258, 33.319, 118.778, 17.56]
  MoveL 10440 to (238.89, 43.33, 144.49) mm, rotated rx 180 ry 0 rz 180 deg; joints [-28.78, 58.941, -92.258, 33.319, 118.778, 17.56]
  Call Extruder(596.44861)
  MoveL 10441 to (239, 43.58, 144.49) mm, rotated rx -180 ry 0 rz 180 deg; joints [-28.886, 58.966, -92.257, 33.426, 118.725, 17.599]
  MoveL 10442 to (239, 43.58, 144.49) mm, rotated rx -180 ry 0 rz 180 deg; joints [-28.886, 58.966, -92.257, 33.426, 118.725, 17.599]
  Call Extruder(596.60601)
  MoveL 10443 to (239.11, 43.83, 144.49) mm, rotated rx -180 ry 0 rz 180 deg; joints [-28.991, 58.991, -92.256, 33.532, 118.671, 17.638]
  MoveL 10444 to (239.11, 43.83, 144.49) mm, rotated rx -180 ry 0 rz 180 deg; joints [-28.991, 58.991, -92.256, 33.532, 118.671, 17.638]
  Call Extruder(596.78872)
  MoveL 10445 to (239.22, 44.12, 144.49) mm, rotated rx -180 ry 0 rz 180 deg; joints [-29.116, 59.02, -92.254, 33.659, 118.608, 17.684]
  MoveL 10446 to (239.22, 44.12, 144.49) mm, rotated rx -180 ry 0 rz 180 deg; joints [-29.116, 59.02, -92.254, 33.659, 118.608, 17.684]
  Call Extruder(596.97068)
  MoveL 10447 to (239.35, 44.42, 144.49) mm, rotated rx -180 ry 0 rz -180 deg; joints [-29.24, 59.048, -92.253, 33.783, 118.545, 17.729]
  MoveL 10448 to (239.35, 44.42, 144.49) mm, rotated rx -180 ry 0 rz -180 deg; joints [-29.24, 59.048, -92.253, 33.783, 118.545, 17.729]
  Call Extruder(597.11801)
  MoveL 10449 to (239.44, 44.66, 144.49) mm, rotated rx 180 ry 0 rz -180 deg; joints [-29.343, 59.071, -92.251, 33.889, 118.493, 17.767]
  MoveL 10450 to (239.44, 44.66, 144.49) mm, rotated rx 180 ry 0 rz -180 deg; joints [-29.343, 59.071, -92.251, 33.889, 118.493, 17.767]
  Call Extruder(597.23124)
  MoveL 10451 to (239.5, 44.85, 144.49) mm, rotated rx -180 ry 0 rz -180 deg; joints [-29.428, 59.088, -92.25, 33.975, 118.453, 17.799]
  MoveL 10452 to (239.5, 44.85, 144.49) mm, rotated rx -180 ry 0 rz -180 deg; joints [-29.428, 59.088, -92.25, 33.975, 118.453, 17.799]
  Call Extruder(597.34404)
  MoveL 10453 to (239.56, 45.03, 144.49) mm, rotated rx 180 ry 0 rz 180 deg; joints [-29.512, 59.105, -92.249, 34.06, 118.412, 17.831]
  MoveL 10454 to (239.56, 45.03, 144.49) mm, rotated rx 180 ry 0 rz 180 deg; joints [-29.512, 59.105, -92.249, 34.06, 118.412, 17.831]
  Call Extruder(597.45638)
  MoveL 10455 to (239.62, 45.22, 144.49) mm, rotated rx 180 ry 0 rz 180 deg; joints [-29.596, 59.122, -92.248, 34.145, 118.372, 17.863]
  MoveL 10456 to (239.62, 45.22, 144.49) mm, rotated rx 180 ry 0 rz 180 deg; joints [-29.596, 59.122, -92.248, 34.145, 118.372, 17.863]
  Call Extruder(597.56829)
  MoveL 10457 to (239.68, 45.41, 144.49) mm, rotated rx -180 ry 0 rz 180 deg; joints [-29.679, 59.139, -92.248, 34.23, 118.331, 17.894]
  MoveL 10458 to (239.68, 45.41, 144.49) mm, rotated rx -180 ry 0 rz 180 deg; joints [-29.679, 59.139, -92.248, 34.23, 118.331, 17.894]
  Call Extruder(597.68969)
  MoveL 10459 to (239.75, 45.62, 144.49) mm, rotated rx -180 ry 0 rz 180 deg; joints [-29.77, 59.158, -92.246, 34.323, 118.287, 17.929]
  MoveL 10460 to (239.75, 45.62, 144.49) mm, rotated rx -180 ry 0 rz 180 deg; joints [-29.77, 59.158, -92.246, 34.323, 118.287, 17.929]
  Call Extruder(597.82048)
  MoveL 10461 to (239.82, 45.84, 144.49) mm, rotated rx 180 ry 0 rz 180 deg; joints [-29.871, 59.177, -92.245, 34.425, 118.239, 17.966]
  MoveL 10462 to (239.82, 45.84, 144.49) mm, rotated rx 180 ry 0 rz 180 deg; joints [-29.871, 59.177, -92.245, 34.425, 118.239, 17.966]
  Call Extruder(597.95070)
  MoveL 10463 to (239.88, 46.06, 144.49) mm, rotated rx -180 ry 0 rz 180 deg; joints [-29.97, 59.197, -92.244, 34.526, 118.191, 18.004]
  MoveL 10464 to (239.88, 46.06, 144.49) mm, rotated rx -180 ry 0 rz 180 deg; joints [-29.97, 59.197, -92.244, 34.526, 118.191, 18.004]
  Call Extruder(598.08036)
  MoveL 10465 to (239.95, 46.29, 144.49) mm, rotated rx 180 ry 0 rz 180 deg; joints [-30.069, 59.217, -92.243, 34.627, 118.143, 18.041]
  MoveL 10466 to (239.95, 46.29, 144.49) mm, rotated rx 180 ry 0 rz 180 deg; joints [-30.069, 59.217, -92.243, 34.627, 118.143, 18.041]
  Call Extruder(598.20946)
  MoveL 10467 to (240.02, 46.51, 144.49) mm, rotated rx -180 ry 0 rz 180 deg; joints [-30.168, 59.237, -92.242, 34.727, 118.095, 18.078]
  MoveL 10468 to (240.02, 46.51, 144.49) mm, rotated rx -180 ry 0 rz 180 deg; joints [-30.168, 59.237, -92.242, 34.727, 118.095, 18.078]
  Call Extruder(598.32451)
  MoveL 10469 to (240.06, 46.72, 144.49) mm, rotated rx -180 ry 0 rz 180 deg; joints [-30.263, 59.253, -92.241, 34.824, 118.051, 18.115]
  MoveL 10470 to (240.06, 46.72, 144.49) mm, rotated rx -180 ry 0 rz 180 deg; joints [-30.263, 59.253, -92.241, 34.824, 118.051, 18.115]
  Call Extruder(598.43912)
  MoveL 10471 to (240.11, 46.92, 144.49) mm, rotated rx 180 ry 0 rz 180 deg; joints [-30.358, 59.269, -92.24, 34.921, 118.008, 18.151]
  MoveL 10472 to (240.11, 46.92, 144.49) mm, rotated rx 180 ry 0 rz 180 deg; joints [-30.358, 59.269, -92.24, 34.921, 118.008, 18.151]
  Call Extruder(598.55327)
  MoveL 10473 to (240.15, 47.12, 144.49) mm, rotated rx 180 ry 0 rz 180 deg; joints [-30.453, 59.286, -92.239, 35.018, 117.964, 18.188]
  MoveL 10474 to (240.15, 47.12, 144.49) mm, rotated rx 180 ry 0 rz 180 deg; joints [-30.453, 59.286, -92.239, 35.018, 117.964, 18.188]
  Call Extruder(598.66696)
  MoveL 10475 to (240.2, 47.33, 144.49) mm, rotated rx -180 ry 0 rz 180 deg; joints [-30.548, 59.302, -92.238, 35.114, 117.92, 18.224]
  MoveL 10476 to (240.2, 47.33, 144.49) mm, rotated rx -180 ry 0 rz 180 deg; joints [-30.548, 59.302, -92.238, 35.114, 117.92, 18.224]
  Call Extruder(598.79237)
  MoveL 10477 to (240.24, 47.56, 144.49) mm, rotated rx 180 ry 0 rz 180 deg; joints [-30.653, 59.32, -92.237, 35.221, 117.871, 18.265]
  MoveL 10478 to (240.24, 47.56, 144.49) mm, rotated rx 180 ry 0 rz 180 deg; joints [-30.653, 59.32, -92.237, 35.221, 117.871, 18.265]
  Call Extruder(598.92935)
  MoveL 10479 to (240.29, 47.8, 144.49) mm, rotated rx -180 ry 0 rz 180 deg; joints [-30.768, 59.34, -92.236, 35.339, 117.818, 18.309]
  MoveL 10480 to (240.29, 47.8, 144.49) mm, rotated rx -180 ry 0 rz 180 deg; joints [-30.768, 59.34, -92.236, 35.339, 117.818, 18.309]
  Call Extruder(599.06572)
  MoveL 10481 to (240.34, 48.05, 144.49) mm, rotated rx -180 ry 0 rz 180 deg; joints [-30.884, 59.36, -92.234, 35.457, 117.765, 18.353]
  MoveL 10482 to (240.34, 48.05, 144.49) mm, rotated rx -180 ry 0 rz 180 deg; joints [-30.884, 59.36, -92.234, 35.457, 117.765, 18.353]
  Call Extruder(599.20147)
  MoveL 10483 to (240.39, 48.3, 144.49) mm, rotated rx -180 ry 0 rz 180 deg; joints [-30.999, 59.379, -92.233, 35.574, 117.711, 18.397]
  MoveL 10484 to (240.39, 48.3, 144.49) mm, rotated rx -180 ry 0 rz 180 deg; joints [-30.999, 59.379, -92.233, 35.574, 117.711, 18.397]
  Call Extruder(599.33662)
  MoveL 10485 to (240.44, 48.55, 144.49) mm, rotated rx -180 ry 0 rz 180 deg; joints [-31.114, 59.399, -92.232, 35.69, 117.658, 18.44]
  MoveL 10486 to (240.44, 48.55, 144.49) mm, rotated rx -180 ry 0 rz 180 deg; joints [-31.114, 59.399, -92.232, 35.69, 117.658, 18.44]
  Call Extruder(599.47116)
  MoveL 10487 to (240.49, 48.8, 144.49) mm, rotated rx -180 ry 0 rz 180 deg; joints [-31.228, 59.419, -92.231, 35.806, 117.605, 18.483]
  MoveL 10488 to (240.49, 48.8, 144.49) mm, rotated rx -180 ry 0 rz 180 deg; joints [-31.228, 59.419, -92.231, 35.806, 117.605, 18.483]
  Call Extruder(599.60508)
  MoveL 10489 to (240.54, 49.05, 144.49) mm, rotated rx -180 ry 0 rz 180 deg; joints [-31.342, 59.439, -92.229, 35.922, 117.551, 18.526]
  MoveL 10490 to (240.54, 49.05, 144.49) mm, rotated rx -180 ry 0 rz 180 deg; joints [-31.342, 59.439, -92.229, 35.922, 117.551, 18.526]
  Call Extruder(599.75295)
  MoveL 10491 to (240.59, 49.33, 144.49) mm, rotated rx -180 ry 0 rz 180 deg; joints [-31.47, 59.46, -92.228, 36.051, 117.492, 18.574]
  MoveL 10492 to (240.59, 49.33, 144.49) mm, rotated rx -180 ry 0 rz 180 deg; joints [-31.47, 59.46, -92.228, 36.051, 117.492, 18.574]
  Call Extruder(599.91470)
  MoveL 10493 to (240.64, 49.63, 144.49) mm, rotated rx 180 ry 0 rz 180 deg; joints [-31.612, 59.483, -92.226, 36.196, 117.427, 18.627]
  MoveL 10494 to (240.64, 49.63, 144.49) mm, rotated rx 180 ry 0 rz 180 deg; joints [-31.612, 59.483, -92.226, 36.196, 117.427, 18.627]
  Call Extruder(600.07571)
  MoveL 10495 to (240.69, 49.94, 144.49) mm, rotated rx -180 ry 0 rz 180 deg; joints [-31.755, 59.507, -92.225, 36.34, 117.361, 18.681]
  MoveL 10496 to (240.69, 49.94, 144.49) mm, rotated rx -180 ry 0 rz 180 deg; joints [-31.755, 59.507, -92.225, 36.34, 117.361, 18.681]
  Call Extruder(600.23600)
  MoveL 10497 to (240.74, 50.24, 144.49) mm, rotated rx -180 ry 0 rz 180 deg; joints [-31.895, 59.53, -92.223, 36.482, 117.296, 18.733]
  MoveL 10498 to (240.74, 50.24, 144.49) mm, rotated rx -180 ry 0 rz 180 deg; joints [-31.895, 59.53, -92.223, 36.482, 117.296, 18.733]
  Call Extruder(600.39556)
  MoveL 10499 to (240.78, 50.55, 144.49) mm, rotated rx -180 ry 0 rz 180 deg; joints [-32.036, 59.553, -92.222, 36.625, 117.231, 18.785]
  MoveL 10500 to (240.78, 50.55, 144.49) mm, rotated rx -180 ry 0 rz 180 deg; joints [-32.036, 59.553, -92.222, 36.625, 117.231, 18.785]
  Call Extruder(600.55440)
  MoveL 10501 to (240.83, 50.86, 144.49) mm, rotated rx 180 ry 0 rz 180 deg; joints [-32.176, 59.577, -92.22, 36.766, 117.165, 18.836]
  MoveL 10502 to (240.83, 50.86, 144.49) mm, rotated rx 180 ry 0 rz 180 deg; joints [-32.176, 59.577, -92.22, 36.766, 117.165, 18.836]
  Call Extruder(600.73307)
  MoveL 10503 to (240.88, 51.2, 144.49) mm, rotated rx -180 ry 0 rz 180 deg; joints [-32.337, 59.603, -92.218, 36.928, 117.091, 18.895]
  MoveL 10504 to (240.88, 51.2, 144.49) mm, rotated rx -180 ry 0 rz 180 deg; joints [-32.337, 59.603, -92.218, 36.928, 117.091, 18.895]
  Call Extruder(600.93151)
  MoveL 10505 to (240.93, 51.59, 144.49) mm, rotated rx 180 ry 0 rz -180 deg; joints [-32.518, 59.631, -92.216, 37.111, 117.008, 18.962]
  MoveL 10506 to (240.93, 51.59, 144.49) mm, rotated rx 180 ry 0 rz -180 deg; joints [-32.518, 59.631, -92.216, 37.111, 117.008, 18.962]
  Call Extruder(601.12909)
  MoveL 10507 to (240.97, 51.98, 144.49) mm, rotated rx 180 ry 0 rz 180 deg; joints [-32.697, 59.659, -92.214, 37.292, 116.926, 19.028]
  MoveL 10508 to (240.97, 51.98, 144.49) mm, rotated rx 180 ry 0 rz 180 deg; joints [-32.697, 59.659, -92.214, 37.292, 116.926, 19.028]
  Call Extruder(601.32579)
  MoveL 10509 to (241.02, 52.36, 144.49) mm, rotated rx -180 ry 0 rz 180 deg; joints [-32.876, 59.688, -92.212, 37.473, 116.843, 19.093]
  MoveL 10510 to (241.02, 52.36, 144.49) mm, rotated rx -180 ry 0 rz 180 deg; joints [-32.876, 59.688, -92.212, 37.473, 116.843, 19.093]
  Call Extruder(601.52163)
  MoveL 10511 to (241.06, 52.75, 144.49) mm, rotated rx 180 ry 0 rz 180 deg; joints [-33.055, 59.717, -92.21, 37.652, 116.76, 19.157]
  MoveL 10512 to (241.06, 52.75, 144.49) mm, rotated rx 180 ry 0 rz 180 deg; joints [-33.055, 59.717, -92.21, 37.652, 116.76, 19.157]
  Call Extruder(601.81707)
  MoveL 10513 to (241.11, 53.34, 144.49) mm, rotated rx -180 ry 0 rz 180 deg; joints [-33.331, 59.758, -92.207, 37.93, 116.634, 19.258]
  MoveL 10514 to (241.11, 53.34, 144.49) mm, rotated rx -180 ry 0 rz 180 deg; joints [-33.331, 59.758, -92.207, 37.93, 116.634, 19.258]
  Call Extruder(602.11118)
  MoveL 10515 to (241.16, 53.93, 144.49) mm, rotated rx 180 ry 0 rz 180 deg; joints [-33.606, 59.8, -92.204, 38.206, 116.508, 19.356]
  MoveL 10516 to (241.16, 53.93, 144.49) mm, rotated rx 180 ry 0 rz 180 deg; joints [-33.606, 59.8, -92.204, 38.206, 116.508, 19.356]
  Call Extruder(602.40395)
  MoveL 10517 to (241.2, 54.52, 144.49) mm, rotated rx 180 ry 0 rz 180 deg; joints [-33.878, 59.842, -92.2, 38.48, 116.382, 19.453]
  MoveL 10518 to (241.2, 54.52, 144.49) mm, rotated rx 180 ry 0 rz 180 deg; joints [-33.878, 59.842, -92.2, 38.48, 116.382, 19.453]
  Call Extruder(602.97740)
  MoveL 10519 to (241.25, 55.68, 144.49) mm, rotated rx 180 ry 0 rz 180 deg; joints [-34.425, 59.921, -92.194, 39.027, 116.132, 19.647]
  MoveL 10520 to (241.25, 55.68, 144.49) mm, rotated rx 180 ry 0 rz 180 deg; joints [-34.425, 59.921, -92.194, 39.027, 116.132, 19.647]
  Call Extruder(603.69124)
  MoveL 10521 to (241.29, 57.14, 144.49) mm, rotated rx 180 ry 0 rz 180 deg; joints [-35.104, 60.019, -92.186, 39.705, 115.82, 19.884]
  Call Extruder(645.75613)
  MoveL 10522 to (241.29, 142.86, 144.49) mm, rotated rx -180 ry 0 rz 180 deg; joints [-60.361, 66.861, -90.745, 62.514, 101.55, 21.05]
  Call Extruder(646.18456)
  MoveL 10523 to (241.27, 143.74, 144.49) mm, rotated rx 180 ry 0 rz 180 deg; joints [-60.516, 66.933, -90.718, 62.643, 101.45, 20.99]
  MoveL 10524 to (241.27, 143.74, 144.49) mm, rotated rx 180 ry 0 rz 180 deg; joints [-60.516, 66.933, -90.718, 62.643, 101.45, 20.99]
  Call Extruder(646.75801)
  MoveL 10525 to (241.23, 144.9, 144.49) mm, rotated rx 180 ry 0 rz 180 deg; joints [-60.726, 67.027, -90.683, 62.821, 101.315, 20.912]
  MoveL 10526 to (241.23, 144.9, 144.49) mm, rotated rx 180 ry 0 rz 180 deg; joints [-60.726, 67.027, -90.683, 62.821, 101.315, 20.912]
  Call Extruder(647.19234)
  MoveL 10527 to (241.18, 145.77, 144.49) mm, rotated rx 180 ry 0 rz -180 deg; joints [-60.887, 67.098, -90.657, 62.957, 101.213, 20.854]
  MoveL 10528 to (241.18, 145.77, 144.49) mm, rotated rx 180 ry 0 rz -180 deg; joints [-60.887, 67.098, -90.657, 62.957, 101.213, 20.854]
  Call Extruder(647.48645)
  MoveL 10529 to (241.13, 146.36, 144.49) mm, rotated rx 180 ry 0 rz 180 deg; joints [-61, 67.145, -90.639, 63.053, 101.144, 20.817]
  MoveL 10530 to (241.13, 146.36, 144.49) mm, rotated rx 180 ry 0 rz 180 deg; joints [-61, 67.145, -90.639, 63.053, 101.144, 20.817]
  Call Extruder(647.78189)
  MoveL 10531 to (241.09, 146.95, 144.49) mm, rotated rx -180 ry 0 rz -180 deg; joints [-61.111, 67.192, -90.622, 63.148, 101.075, 20.778]
  MoveL 10532 to (241.09, 146.95, 144.49) mm, rotated rx -180 ry 0 rz -180 deg; joints [-61.111, 67.192, -90.622, 63.148, 101.075, 20.778]
  Call Extruder(648.02815)
  MoveL 10533 to (241.04, 147.44, 144.49) mm, rotated rx 180 ry 0 rz 180 deg; joints [-61.205, 67.23, -90.607, 63.228, 101.018, 20.747]
  MoveL 10534 to (241.04, 147.44, 144.49) mm, rotated rx 180 ry 0 rz 180 deg; joints [-61.205, 67.23, -90.607, 63.228, 101.018, 20.747]
  Call Extruder(648.22485)
  MoveL 10535 to (240.99, 147.83, 144.49) mm, rotated rx 180 ry 0 rz 180 deg; joints [-61.282, 67.26, -90.596, 63.294, 100.972, 20.724]
  MoveL 10536 to (240.99, 147.83, 144.49) mm, rotated rx 180 ry 0 rz 180 deg; joints [-61.282, 67.26, -90.596, 63.294, 100.972, 20.724]
  Call Extruder(648.42243)
  MoveL 10537 to (240.95, 148.22, 144.49) mm, rotated rx -180 ry 0 rz 180 deg; joints [-61.359, 67.29, -90.584, 63.36, 100.926, 20.7]
  MoveL 10538 to (240.95, 148.22, 144.49) mm, rotated rx -180 ry 0 rz 180 deg; joints [-61.359, 67.29, -90.584, 63.36, 100.926, 20.7]
  Call Extruder(648.62087)
  MoveL 10539 to (240.9, 148.6, 144.49) mm, rotated rx -180 ry 0 rz 180 deg; joints [-61.436, 67.32, -90.572, 63.426, 100.881, 20.676]
  MoveL 10540 to (240.9, 148.6, 144.49) mm, rotated rx -180 ry 0 rz 180 deg; joints [-61.436, 67.32, -90.572, 63.426, 100.881, 20.676]
  Call Extruder(648.82018)
  MoveL 10541 to (240.86, 148.99, 144.49) mm, rotated rx 180 ry 0 rz -180 deg; joints [-61.512, 67.35, -90.561, 63.492, 100.835, 20.651]
  MoveL 10542 to (240.86, 148.99, 144.49) mm, rotated rx 180 ry 0 rz -180 deg; joints [-61.512, 67.35, -90.561, 63.492, 100.835, 20.651]
  Call Extruder(648.97901)
  MoveL 10543 to (240.81, 149.3, 144.49) mm, rotated rx -180 ry 0 rz 180 deg; joints [-61.575, 67.373, -90.552, 63.547, 100.798, 20.633]
  MoveL 10544 to (240.81, 149.3, 144.49) mm, rotated rx -180 ry 0 rz 180 deg; joints [-61.575, 67.373, -90.552, 63.547, 100.798, 20.633]
  Call Extruder(649.13857)
  MoveL 10545 to (240.76, 149.6, 144.49) mm, rotated rx 180 ry 0 rz 180 deg; joints [-61.639, 67.396, -90.543, 63.602, 100.762, 20.615]
  MoveL 10546 to (240.76, 149.6, 144.49) mm, rotated rx 180 ry 0 rz 180 deg; joints [-61.639, 67.396, -90.543, 63.602, 100.762, 20.615]
  Call Extruder(649.29886)
  MoveL 10547 to (240.71, 149.91, 144.49) mm, rotated rx -180 ry 0 rz 180 deg; joints [-61.702, 67.419, -90.533, 63.656, 100.725, 20.597]
  MoveL 10548 to (240.71, 149.91, 144.49) mm, rotated rx -180 ry 0 rz 180 deg; joints [-61.702, 67.419, -90.533, 63.656, 100.725, 20.597]
  Call Extruder(649.45987)
  MoveL 10549 to (240.66, 150.21, 144.49) mm, rotated rx -180 ry 0 rz 180 deg; joints [-61.765, 67.442, -90.524, 63.711, 100.689, 20.579]
  MoveL 10550 to (240.66, 150.21, 144.49) mm, rotated rx -180 ry 0 rz 180 deg; joints [-61.765, 67.442, -90.524, 63.711, 100.689, 20.579]
  Call Extruder(649.62162)
  MoveL 10551 to (240.61, 150.52, 144.49) mm, rotated rx 180 ry 0 rz 180 deg; joints [-61.828, 67.466, -90.515, 63.765, 100.652, 20.561]
  MoveL 10552 to (240.61, 150.52, 144.49) mm, rotated rx 180 ry 0 rz 180 deg; joints [-61.828, 67.466, -90.515, 63.765, 100.652, 20.561]
  Call Extruder(649.78409)
  MoveL 10553 to (240.57, 150.83, 144.49) mm, rotated rx 180 ry 0 rz 180 deg; joints [-61.891, 67.489, -90.506, 63.82, 100.616, 20.542]
  MoveL 10554 to (240.57, 150.83, 144.49) mm, rotated rx 180 ry 0 rz 180 deg; joints [-61.891, 67.489, -90.506, 63.82, 100.616, 20.542]
  Call Extruder(649.91802)
  MoveL 10555 to (240.52, 151.08, 144.49) mm, rotated rx 180 ry 0 rz -180 deg; joints [-61.944, 67.507, -90.499, 63.867, 100.586, 20.528]
  MoveL 10556 to (240.52, 151.08, 144.49) mm, rotated rx 180 ry 0 rz -180 deg; joints [-61.944, 67.507, -90.499, 63.867, 100.586, 20.528]
  Call Extruder(650.05255)
  MoveL 10557 to (240.47, 151.32, 144.49) mm, rotated rx -180 ry 0 rz 180 deg; joints [-61.998, 67.525, -90.491, 63.914, 100.556, 20.514]
  MoveL 10558 to (240.47, 151.32, 144.49) mm, rotated rx -180 ry 0 rz 180 deg; joints [-61.998, 67.525, -90.491, 63.914, 100.556, 20.514]
  Call Extruder(650.18770)
  MoveL 10559 to (240.42, 151.57, 144.49) mm, rotated rx 180 ry 0 rz 180 deg; joints [-62.052, 67.544, -90.484, 63.961, 100.525, 20.5]
  MoveL 10560 to (240.42, 151.57, 144.49) mm, rotated rx 180 ry 0 rz 180 deg; joints [-62.052, 67.544, -90.484, 63.961, 100.525, 20.5]
  Call Extruder(650.32346)
  MoveL 10561 to (240.37, 151.82, 144.49) mm, rotated rx -180 ry 0 rz 180 deg; joints [-62.105, 67.562, -90.477, 64.007, 100.495, 20.486]
  MoveL 10562 to (240.37, 151.82, 144.49) mm, rotated rx -180 ry 0 rz 180 deg; joints [-62.105, 67.562, -90.477, 64.007, 100.495, 20.486]
  Call Extruder(650.45983)
  MoveL 10563 to (240.32, 152.07, 144.49) mm, rotated rx 180 ry 0 rz 180 deg; joints [-62.159, 67.581, -90.469, 64.054, 100.465, 20.471]
  MoveL 10564 to (240.32, 152.07, 144.49) mm, rotated rx 180 ry 0 rz 180 deg; joints [-62.159, 67.581, -90.469, 64.054, 100.465, 20.471]
  Call Extruder(650.59680)
  MoveL 10565 to (240.27, 152.32, 144.49) mm, rotated rx 180 ry 0 rz -180 deg; joints [-62.212, 67.599, -90.462, 64.1, 100.436, 20.457]
  MoveL 10566 to (240.27, 152.32, 144.49) mm, rotated rx 180 ry 0 rz -180 deg; joints [-62.212, 67.599, -90.462, 64.1, 100.436, 20.457]
  Call Extruder(650.73439)
  MoveL 10567 to (240.22, 152.57, 144.49) mm, rotated rx 180 ry 0 rz -180 deg; joints [-62.265, 67.617, -90.454, 64.147, 100.406, 20.442]
  MoveL 10568 to (240.22, 152.57, 144.49) mm, rotated rx 180 ry 0 rz -180 deg; joints [-62.265, 67.617, -90.454, 64.147, 100.406, 20.442]
  Call Extruder(650.84809)
  MoveL 10569 to (240.17, 152.77, 144.49) mm, rotated rx 180 ry 0 rz 180 deg; joints [-62.31, 67.632, -90.448, 64.186, 100.381, 20.431]
  MoveL 10570 to (240.17, 152.77, 144.49) mm, rotated rx 180 ry 0 rz 180 deg; joints [-62.31, 67.632, -90.448, 64.186, 100.381, 20.431]
  Call Extruder(650.96224)
  MoveL 10571 to (240.13, 152.98, 144.49) mm, rotated rx 180 ry 0 rz -180 deg; joints [-62.355, 67.647, -90.442, 64.225, 100.356, 20.419]
  MoveL 10572 to (240.13, 152.98, 144.49) mm, rotated rx 180 ry 0 rz -180 deg; joints [-62.355, 67.647, -90.442, 64.225, 100.356, 20.419]
  Call Extruder(651.07684)
  MoveL 10573 to (240.08, 153.18, 144.49) mm, rotated rx -180 ry 0 rz 180 deg; joints [-62.399, 67.662, -90.436, 64.264, 100.332, 20.408]
  MoveL 10574 to (240.08, 153.18, 144.49) mm, rotated rx -180 ry 0 rz 180 deg; joints [-62.399, 67.662, -90.436, 64.264, 100.332, 20.408]
  Call Extruder(651.19190)
  MoveL 10575 to (240.04, 153.39, 144.49) mm, rotated rx -180 ry 0 rz 180 deg; joints [-62.444, 67.677, -90.43, 64.303, 100.307, 20.396]
  MoveL 10576 to (240.04, 153.39, 144.49) mm, rotated rx -180 ry 0 rz 180 deg; joints [-62.444, 67.677, -90.43, 64.303, 100.307, 20.396]
  Call Extruder(651.31412)
  MoveL 10577 to (239.98, 153.6, 144.49) mm, rotated rx -180 ry 0 rz 180 deg; joints [-62.493, 67.692, -90.424, 64.346, 100.281, 20.385]
  MoveL 10578 to (239.98, 153.6, 144.49) mm, rotated rx -180 ry 0 rz 180 deg; joints [-62.493, 67.692, -90.424, 64.346, 100.281, 20.385]
  Call Extruder(651.44378)
  MoveL 10579 to (239.92, 153.82, 144.49) mm, rotated rx -180 ry 0 rz -180 deg; joints [-62.547, 67.708, -90.417, 64.394, 100.252, 20.374]
  MoveL 10580 to (239.92, 153.82, 144.49) mm, rotated rx -180 ry 0 rz -180 deg; joints [-62.547, 67.708, -90.417, 64.394, 100.252, 20.374]
  Call Extruder(651.57401)
  MoveL 10581 to (239.85, 154.05, 144.49) mm, rotated rx 180 ry 0 rz 180 deg; joints [-62.601, 67.723, -90.411, 64.442, 100.224, 20.363]
  MoveL 10582 to (239.85, 154.05, 144.49) mm, rotated rx 180 ry 0 rz 180 deg; joints [-62.601, 67.723, -90.411, 64.442, 100.224, 20.363]
  Call Extruder(651.70480)
  MoveL 10583 to (239.78, 154.27, 144.49) mm, rotated rx 180 ry 0 rz -180 deg; joints [-62.654, 67.739, -90.405, 64.489, 100.196, 20.352]
  MoveL 10584 to (239.78, 154.27, 144.49) mm, rotated rx 180 ry 0 rz -180 deg; joints [-62.654, 67.739, -90.405, 64.489, 100.196, 20.352]
  Call Extruder(651.83615)
  MoveL 10585 to (239.71, 154.5, 144.49) mm, rotated rx 180 ry 0 rz -180 deg; joints [-62.708, 67.755, -90.398, 64.537, 100.168, 20.34]
  MoveL 10586 to (239.71, 154.5, 144.49) mm, rotated rx 180 ry 0 rz -180 deg; joints [-62.708, 67.755, -90.398, 64.537, 100.168, 20.34]
  Call Extruder(651.94805)
  MoveL 10587 to (239.65, 154.68, 144.49) mm, rotated rx 180 ry 0 rz -180 deg; joints [-62.754, 67.767, -90.393, 64.578, 100.144, 20.332]
  MoveL 10588 to (239.65, 154.68, 144.49) mm, rotated rx 180 ry 0 rz -180 deg; joints [-62.754, 67.767, -90.393, 64.578, 100.144, 20.332]
  Call Extruder(652.06040)
  MoveL 10589 to (239.59, 154.87, 144.49) mm, rotated rx 180 ry 0 rz 180 deg; joints [-62.801, 67.78, -90.387, 64.619, 100.12, 20.322]
  MoveL 10590 to (239.59, 154.87, 144.49) mm, rotated rx 180 ry 0 rz 180 deg; joints [-62.801, 67.78, -90.387, 64.619, 100.12, 20.322]
  Call Extruder(652.17319)
  MoveL 10591 to (239.53, 155.06, 144.49) mm, rotated rx -180 ry 0 rz 180 deg; joints [-62.847, 67.793, -90.382, 64.66, 100.096, 20.313]
  MoveL 10592 to (239.53, 155.06, 144.49) mm, rotated rx -180 ry 0 rz 180 deg; joints [-62.847, 67.793, -90.382, 64.66, 100.096, 20.313]
  Call Extruder(652.28642)
  MoveL 10593 to (239.47, 155.25, 144.49) mm, rotated rx -180 ry 0 rz 180 deg; joints [-62.893, 67.806, -90.377, 64.701, 100.072, 20.304]
  MoveL 10594 to (239.47, 155.25, 144.49) mm, rotated rx -180 ry 0 rz 180 deg; joints [-62.893, 67.806, -90.377, 64.701, 100.072, 20.304]
  Call Extruder(652.40010)
  MoveL 10595 to (239.41, 155.44, 144.49) mm, rotated rx 180 ry 0 rz -180 deg; joints [-62.939, 67.819, -90.371, 64.742, 100.048, 20.295]
  MoveL 10596 to (239.41, 155.44, 144.49) mm, rotated rx 180 ry 0 rz -180 deg; joints [-62.939, 67.819, -90.371, 64.742, 100.048, 20.295]
  Call Extruder(652.58206)
  MoveL 10597 to (239.29, 155.73, 144.49) mm, rotated rx 180 ry 0 rz 180 deg; joints [-63.018, 67.838, -90.363, 64.813, 100.009, 20.283]
  MoveL 10598 to (239.29, 155.73, 144.49) mm, rotated rx 180 ry 0 rz 180 deg; joints [-63.018, 67.838, -90.363, 64.813, 100.009, 20.283]
  Call Extruder(652.76478)
  MoveL 10599 to (239.17, 156.02, 144.49) mm, rotated rx 180 ry 0 rz 180 deg; joints [-63.097, 67.857, -90.355, 64.884, 99.971, 20.272]
  MoveL 10600 to (239.17, 156.02, 144.49) mm, rotated rx 180 ry 0 rz 180 deg; joints [-63.097, 67.857, -90.355, 64.884, 99.971, 20.272]
  Call Extruder(652.93520)
  MoveL 10601 to (239.05, 156.29, 144.49) mm, rotated rx -180 ry 0 rz -180 deg; joints [-63.17, 67.875, -90.348, 64.949, 99.935, 20.261]
  MoveL 10602 to (239.05, 156.29, 144.49) mm, rotated rx -180 ry 0 rz -180 deg; joints [-63.17, 67.875, -90.348, 64.949, 99.935, 20.261]
  Call Extruder(653.09321)
  MoveL 10603 to (238.94, 156.54, 144.49) mm, rotated rx -180 ry 0 rz -180 deg; joints [-63.238, 67.891, -90.341, 65.01, 99.902, 20.251]
  MoveL 10604 to (238.94, 156.54, 144.49) mm, rotated rx -180 ry 0 rz -180 deg; joints [-63.238, 67.891, -90.341, 65.01, 99.902, 20.251]
  Call Extruder(653.25183)
  MoveL 10605 to (238.84, 156.79, 144.49) mm, rotated rx 180 ry 0 rz -180 deg; joints [-63.306, 67.907, -90.334, 65.072, 99.868, 20.241]
  MoveL 10606 to (238.84, 156.79, 144.49) mm, rotated rx 180 ry 0 rz -180 deg; joints [-63.306, 67.907, -90.334, 65.072, 99.868, 20.241]
  Call Extruder(653.45800)
  MoveL 10607 to (238.66, 157.09, 144.49) mm, rotated rx -180 ry 0 rz -180 deg; joints [-63.401, 67.925, -90.327, 65.159, 99.825, 20.233]
  MoveL 10608 to (238.66, 157.09, 144.49) mm, rotated rx -180 ry 0 rz -180 deg; joints [-63.401, 67.925, -90.327, 65.159, 99.825, 20.233]
  Call Extruder(653.66494)
  MoveL 10609 to (238.49, 157.4, 144.49) mm, rotated rx 180 ry 0 rz 180 deg; joints [-63.497, 67.943, -90.319, 65.246, 99.781, 20.225]
  MoveL 10610 to (238.49, 157.4, 144.49) mm, rotated rx 180 ry 0 rz 180 deg; joints [-63.497, 67.943, -90.319, 65.246, 99.781, 20.225]
  Call Extruder(653.87267)
  MoveL 10611 to (238.31, 157.7, 144.49) mm, rotated rx 180 ry 0 rz 180 deg; joints [-63.592, 67.961, -90.312, 65.332, 99.737, 20.217]
  MoveL 10612 to (238.31, 157.7, 144.49) mm, rotated rx 180 ry 0 rz 180 deg; joints [-63.592, 67.961, -90.312, 65.332, 99.737, 20.217]
  Call Extruder(654.08118)
  MoveL 10613 to (238.14, 158.01, 144.49) mm, rotated rx 180 ry 0 rz 180 deg; joints [-63.687, 67.978, -90.304, 65.419, 99.694, 20.209]
  MoveL 10614 to (238.14, 158.01, 144.49) mm, rotated rx 180 ry 0 rz 180 deg; joints [-63.687, 67.978, -90.304, 65.419, 99.694, 20.209]
  Call Extruder(654.26072)
  MoveL 10615 to (237.96, 158.25, 144.49) mm, rotated rx 180 ry 0 rz 180 deg; joints [-63.774, 67.991, -90.298, 65.498, 99.656, 20.206]
  MoveL 10616 to (237.96, 158.25, 144.49) mm, rotated rx 180 ry 0 rz 180 deg; joints [-63.774, 67.991, -90.298, 65.498, 99.656, 20.206]
  Call Extruder(654.59412)
  MoveL 10617 to (237.63, 158.7, 144.49) mm, rotated rx -180 ry 0 rz 180 deg; joints [-63.934, 68.015, -90.288, 65.645, 99.587, 20.199]
  MoveL 10618 to (237.63, 158.7, 144.49) mm, rotated rx -180 ry 0 rz 180 deg; joints [-63.934, 68.015, -90.288, 65.645, 99.587, 20.199]
  Call Extruder(654.92872)
  MoveL 10619 to (237.3, 159.15, 144.49) mm, rotated rx 180 ry 0 rz 180 deg; joints [-64.094, 68.039, -90.278, 65.792, 99.518, 20.193]
  Call Extruder(655.75669)
  MoveL 10620 to (236.39, 160.19, 144.49) mm, rotated rx 180 ry 0 rz 180 deg; joints [-64.505, 68.089, -90.256, 66.172, 99.347, 20.191]
  Call Extruder(656.58460)
  MoveL 10621 to (235.35, 161.1, 144.49) mm, rotated rx -180 ry 0 rz 180 deg; joints [-64.933, 68.124, -90.241, 66.572, 99.179, 20.21]
  Call Extruder(656.75191)
  MoveL 10622 to (235.13, 161.27, 144.49) mm, rotated rx 180 ry 0 rz 180 deg; joints [-65.021, 68.129, -90.239, 66.655, 99.146, 20.217]
  MoveL 10623 to (235.13, 161.27, 144.49) mm, rotated rx 180 ry 0 rz 180 deg; joints [-65.021, 68.129, -90.239, 66.655, 99.146, 20.217]
  Call Extruder(657.08534)
  MoveL 10624 to (234.68, 161.59, 144.49) mm, rotated rx -180 ry 0 rz 180 deg; joints [-65.197, 68.139, -90.235, 66.82, 99.079, 20.23]
  MoveL 10625 to (234.68, 161.59, 144.49) mm, rotated rx -180 ry 0 rz 180 deg; joints [-65.197, 68.139, -90.235, 66.82, 99.079, 20.23]
  Call Extruder(657.41758)
  MoveL 10626 to (234.22, 161.92, 144.49) mm, rotated rx -180 ry 0 rz -180 deg; joints [-65.374, 68.149, -90.23, 66.986, 99.013, 20.243]
  MoveL 10627 to (234.22, 161.92, 144.49) mm, rotated rx -180 ry 0 rz -180 deg; joints [-65.374, 68.149, -90.23, 66.986, 99.013, 20.243]
  Call Extruder(657.53524)
  MoveL 10628 to (234.05, 162.02, 144.49) mm, rotated rx -180 ry 0 rz 180 deg; joints [-65.437, 68.15, -90.23, 67.045, 98.99, 20.25]
  MoveL 10629 to (234.05, 162.02, 144.49) mm, rotated rx -180 ry 0 rz 180 deg; joints [-65.437, 68.15, -90.23, 67.045, 98.99, 20.25]
  Call Extruder(657.74297)
  MoveL 10630 to (233.75, 162.2, 144.49) mm, rotated rx 180 ry 0 rz -180 deg; joints [-65.549, 68.153, -90.228, 67.152, 98.949, 20.263]
  MoveL 10631 to (233.75, 162.2, 144.49) mm, rotated rx 180 ry 0 rz -180 deg; joints [-65.549, 68.153, -90.228, 67.152, 98.949, 20.263]
  Call Extruder(657.94993)
  MoveL 10632 to (233.45, 162.37, 144.49) mm, rotated rx 180 ry 0 rz 180 deg; joints [-65.662, 68.157, -90.227, 67.257, 98.908, 20.275]
  MoveL 10633 to (233.45, 162.37, 144.49) mm, rotated rx 180 ry 0 rz 180 deg; joints [-65.662, 68.157, -90.227, 67.257, 98.908, 20.275]
  Call Extruder(658.15610)
  MoveL 10634 to (233.14, 162.55, 144.49) mm, rotated rx -180 ry 0 rz 180 deg; joints [-65.774, 68.16, -90.226, 67.363, 98.868, 20.287]
  MoveL 10635 to (233.14, 162.55, 144.49) mm, rotated rx -180 ry 0 rz 180 deg; joints [-65.774, 68.16, -90.226, 67.363, 98.868, 20.287]
  Call Extruder(658.33777)
  MoveL 10636 to (232.87, 162.69, 144.49) mm, rotated rx 180 ry 0 rz 180 deg; joints [-65.874, 68.161, -90.225, 67.458, 98.832, 20.3]
  MoveL 10637 to (232.87, 162.69, 144.49) mm, rotated rx 180 ry 0 rz 180 deg; joints [-65.874, 68.161, -90.225, 67.458, 98.832, 20.3]
  Call Extruder(658.49574)
  MoveL 10638 to (232.62, 162.8, 144.49) mm, rotated rx 180 ry 0 rz 180 deg; joints [-65.961, 68.161, -90.225, 67.541, 98.802, 20.313]
  MoveL 10639 to (232.62, 162.8, 144.49) mm, rotated rx 180 ry 0 rz 180 deg; joints [-65.961, 68.161, -90.225, 67.541, 98.802, 20.313]
  Call Extruder(658.65309)
  MoveL 10640 to (232.37, 162.91, 144.49) mm, rotated rx 180 ry 0 rz 180 deg; joints [-66.048, 68.16, -90.225, 67.623, 98.772, 20.326]
  MoveL 10641 to (232.37, 162.91, 144.49) mm, rotated rx 180 ry 0 rz 180 deg; joints [-66.048, 68.16, -90.225, 67.623, 98.772, 20.326]
  Call Extruder(658.83583)
  MoveL 10642 to (232.07, 163.02, 144.49) mm, rotated rx -180 ry 0 rz -180 deg; joints [-66.149, 68.16, -90.226, 67.72, 98.737, 20.342]
  MoveL 10643 to (232.07, 163.02, 144.49) mm, rotated rx -180 ry 0 rz -180 deg; joints [-66.149, 68.16, -90.226, 67.72, 98.737, 20.342]
  Call Extruder(659.01781)
  MoveL 10644 to (231.78, 163.15, 144.49) mm, rotated rx 180 ry 0 rz 180 deg; joints [-66.251, 68.159, -90.226, 67.816, 98.702, 20.358]
  MoveL 10645 to (231.78, 163.15, 144.49) mm, rotated rx 180 ry 0 rz 180 deg; joints [-66.251, 68.159, -90.226, 67.816, 98.702, 20.358]
  Call Extruder(659.16515)
  MoveL 10646 to (231.54, 163.24, 144.49) mm, rotated rx 180 ry 0 rz 180 deg; joints [-66.333, 68.158, -90.226, 67.895, 98.674, 20.371]
  MoveL 10647 to (231.54, 163.24, 144.49) mm, rotated rx 180 ry 0 rz 180 deg; joints [-66.333, 68.158, -90.226, 67.895, 98.674, 20.371]
  Call Extruder(659.27837)
  MoveL 10648 to (231.35, 163.3, 144.49) mm, rotated rx 180 ry 0 rz 180 deg; joints [-66.397, 68.156, -90.227, 67.955, 98.653, 20.382]
  MoveL 10649 to (231.35, 163.3, 144.49) mm, rotated rx 180 ry 0 rz 180 deg; joints [-66.397, 68.156, -90.227, 67.955, 98.653, 20.382]
  Call Extruder(659.39115)
  MoveL 10650 to (231.17, 163.36, 144.49) mm, rotated rx -180 ry 0 rz 180 deg; joints [-66.46, 68.154, -90.228, 68.016, 98.632, 20.394]
  MoveL 10651 to (231.17, 163.36, 144.49) mm, rotated rx -180 ry 0 rz 180 deg; joints [-66.46, 68.154, -90.228, 68.016, 98.632, 20.394]
  Call Extruder(659.50349)
  MoveL 10652 to (230.98, 163.42, 144.49) mm, rotated rx 180 ry 0 rz -180 deg; joints [-66.524, 68.153, -90.229, 68.076, 98.611, 20.405]
  MoveL 10653 to (230.98, 163.42, 144.49) mm, rotated rx 180 ry 0 rz -180 deg; joints [-66.524, 68.153, -90.229, 68.076, 98.611, 20.405]
  Call Extruder(659.61538)
  MoveL 10654 to (230.79, 163.48, 144.49) mm, rotated rx 180 ry 0 rz -180 deg; joints [-66.587, 68.151, -90.229, 68.137, 98.59, 20.417]
  MoveL 10655 to (230.79, 163.48, 144.49) mm, rotated rx 180 ry 0 rz -180 deg; joints [-66.587, 68.151, -90.229, 68.137, 98.59, 20.417]
  Call Extruder(659.73678)
  MoveL 10656 to (230.58, 163.55, 144.49) mm, rotated rx 180 ry 0 rz 180 deg; joints [-66.656, 68.149, -90.23, 68.203, 98.567, 20.429]
  MoveL 10657 to (230.58, 163.55, 144.49) mm, rotated rx 180 ry 0 rz 180 deg; joints [-66.656, 68.149, -90.23, 68.203, 98.567, 20.429]
  Call Extruder(659.86760)
  MoveL 10658 to (230.36, 163.62, 144.49) mm, rotated rx -180 ry 0 rz -180 deg; joints [-66.731, 68.146, -90.231, 68.274, 98.542, 20.443]
  MoveL 10659 to (230.36, 163.62, 144.49) mm, rotated rx -180 ry 0 rz -180 deg; joints [-66.731, 68.146, -90.231, 68.274, 98.542, 20.443]
  Call Extruder(659.99784)
  MoveL 10660 to (230.14, 163.68, 144.49) mm, rotated rx 180 ry 0 rz 180 deg; joints [-66.805, 68.144, -90.232, 68.345, 98.517, 20.457]
  MoveL 10661 to (230.14, 163.68, 144.49) mm, rotated rx 180 ry 0 rz 180 deg; joints [-66.805, 68.144, -90.232, 68.345, 98.517, 20.457]
  Call Extruder(660.12753)
  MoveL 10662 to (229.91, 163.75, 144.49) mm, rotated rx -180 ry 0 rz 180 deg; joints [-66.88, 68.142, -90.233, 68.416, 98.492, 20.47]
  MoveL 10663 to (229.91, 163.75, 144.49) mm, rotated rx -180 ry 0 rz 180 deg; joints [-66.88, 68.142, -90.233, 68.416, 98.492, 20.47]
  Call Extruder(660.25665)
  MoveL 10664 to (229.69, 163.82, 144.49) mm, rotated rx 180 ry 0 rz 180 deg; joints [-66.955, 68.139, -90.234, 68.488, 98.467, 20.484]
  MoveL 10665 to (229.69, 163.82, 144.49) mm, rotated rx 180 ry 0 rz 180 deg; joints [-66.955, 68.139, -90.234, 68.488, 98.467, 20.484]
  Call Extruder(660.37172)
  MoveL 10666 to (229.48, 163.86, 144.49) mm, rotated rx 180 ry 0 rz 180 deg; joints [-67.021, 68.136, -90.236, 68.551, 98.446, 20.498]
  MoveL 10667 to (229.48, 163.86, 144.49) mm, rotated rx 180 ry 0 rz 180 deg; joints [-67.021, 68.136, -90.236, 68.551, 98.446, 20.498]
  Call Extruder(660.48634)
  MoveL 10668 to (229.28, 163.91, 144.49) mm, rotated rx 180 ry 0 rz 180 deg; joints [-67.087, 68.132, -90.238, 68.614, 98.425, 20.512]
  MoveL 10669 to (229.28, 163.91, 144.49) mm, rotated rx 180 ry 0 rz 180 deg; joints [-67.087, 68.132, -90.238, 68.614, 98.425, 20.512]
  Call Extruder(660.60051)
  MoveL 10670 to (229.08, 163.95, 144.49) mm, rotated rx -180 ry 0 rz 180 deg; joints [-67.153, 68.129, -90.239, 68.677, 98.403, 20.526]
  MoveL 10671 to (229.08, 163.95, 144.49) mm, rotated rx -180 ry 0 rz 180 deg; joints [-67.153, 68.129, -90.239, 68.677, 98.403, 20.526]
  Call Extruder(660.71423)
  MoveL 10672 to (228.87, 164, 144.49) mm, rotated rx 180 ry 0 rz -180 deg; joints [-67.22, 68.125, -90.241, 68.741, 98.382, 20.54]
  MoveL 10673 to (228.87, 164, 144.49) mm, rotated rx 180 ry 0 rz -180 deg; joints [-67.22, 68.125, -90.241, 68.741, 98.382, 20.54]
  Call Extruder(660.83965)
  MoveL 10674 to (228.64, 164.04, 144.49) mm, rotated rx -180 ry 0 rz -180 deg; joints [-67.293, 68.121, -90.242, 68.811, 98.358, 20.555]
  MoveL 10675 to (228.64, 164.04, 144.49) mm, rotated rx -180 ry 0 rz -180 deg; joints [-67.293, 68.121, -90.242, 68.811, 98.358, 20.555]
  Call Extruder(660.97663)
  MoveL 10676 to (228.4, 164.09, 144.49) mm, rotated rx -180 ry 0 rz -180 deg; joints [-67.373, 68.117, -90.244, 68.888, 98.332, 20.572]
  MoveL 10677 to (228.4, 164.09, 144.49) mm, rotated rx -180 ry 0 rz -180 deg; joints [-67.373, 68.117, -90.244, 68.888, 98.332, 20.572]
  Call Extruder(661.11299)
  MoveL 10678 to (228.15, 164.14, 144.49) mm, rotated rx 180 ry 0 rz 180 deg; joints [-67.453, 68.112, -90.246, 68.965, 98.307, 20.59]
  MoveL 10679 to (228.15, 164.14, 144.49) mm, rotated rx 180 ry 0 rz 180 deg; joints [-67.453, 68.112, -90.246, 68.965, 98.307, 20.59]
  Call Extruder(661.24875)
  MoveL 10680 to (227.9, 164.19, 144.49) mm, rotated rx 180 ry 0 rz 180 deg; joints [-67.534, 68.108, -90.248, 69.042, 98.281, 20.607]
  MoveL 10681 to (227.9, 164.19, 144.49) mm, rotated rx 180 ry 0 rz 180 deg; joints [-67.534, 68.108, -90.248, 69.042, 98.281, 20.607]
  Call Extruder(661.38390)
  MoveL 10682 to (227.65, 164.24, 144.49) mm, rotated rx -180 ry 0 rz 180 deg; joints [-67.614, 68.103, -90.25, 69.119, 98.255, 20.624]
  MoveL 10683 to (227.65, 164.24, 144.49) mm, rotated rx -180 ry 0 rz 180 deg; joints [-67.614, 68.103, -90.25, 69.119, 98.255, 20.624]
  Call Extruder(661.51844)
  MoveL 10684 to (227.4, 164.29, 144.49) mm, rotated rx -180 ry 0 rz 180 deg; joints [-67.695, 68.099, -90.252, 69.195, 98.229, 20.641]
  MoveL 10685 to (227.4, 164.29, 144.49) mm, rotated rx -180 ry 0 rz 180 deg; joints [-67.695, 68.099, -90.252, 69.195, 98.229, 20.641]
  Call Extruder(661.65236)
  MoveL 10686 to (227.15, 164.34, 144.49) mm, rotated rx 180 ry 0 rz -180 deg; joints [-67.775, 68.094, -90.254, 69.272, 98.203, 20.658]
  MoveL 10687 to (227.15, 164.34, 144.49) mm, rotated rx 180 ry 0 rz -180 deg; joints [-67.775, 68.094, -90.254, 69.272, 98.203, 20.658]
  Call Extruder(661.80023)
  MoveL 10688 to (226.87, 164.39, 144.49) mm, rotated rx 180 ry 0 rz 180 deg; joints [-67.864, 68.089, -90.257, 69.357, 98.174, 20.677]
  MoveL 10689 to (226.87, 164.39, 144.49) mm, rotated rx 180 ry 0 rz 180 deg; joints [-67.864, 68.089, -90.257, 69.357, 98.174, 20.677]
  Call Extruder(661.96197)
  MoveL 10690 to (226.57, 164.44, 144.49) mm, rotated rx 180 ry 0 rz -180 deg; joints [-67.961, 68.082, -90.259, 69.451, 98.143, 20.699]
  MoveL 10691 to (226.57, 164.44, 144.49) mm, rotated rx 180 ry 0 rz -180 deg; joints [-67.961, 68.082, -90.259, 69.451, 98.143, 20.699]
  Call Extruder(662.12298)
  MoveL 10692 to (226.26, 164.49, 144.49) mm, rotated rx 180 ry 0 rz -180 deg; joints [-68.059, 68.076, -90.262, 69.544, 98.112, 20.72]
  MoveL 10693 to (226.26, 164.49, 144.49) mm, rotated rx 180 ry 0 rz -180 deg; joints [-68.059, 68.076, -90.262, 69.544, 98.112, 20.72]
  Call Extruder(662.28327)
  MoveL 10694 to (225.96, 164.54, 144.49) mm, rotated rx 180 ry 0 rz 180 deg; joints [-68.156, 68.07, -90.265, 69.637, 98.08, 20.742]
  MoveL 10695 to (225.96, 164.54, 144.49) mm, rotated rx 180 ry 0 rz 180 deg; joints [-68.156, 68.07, -90.265, 69.637, 98.08, 20.742]
  Call Extruder(662.44282)
  MoveL 10696 to (225.65, 164.58, 144.49) mm, rotated rx 180 ry 0 rz 180 deg; joints [-68.254, 68.063, -90.268, 69.73, 98.049, 20.763]
  MoveL 10697 to (225.65, 164.58, 144.49) mm, rotated rx 180 ry 0 rz 180 deg; joints [-68.254, 68.063, -90.268, 69.73, 98.049, 20.763]
  Call Extruder(662.60165)
  MoveL 10698 to (225.34, 164.63, 144.49) mm, rotated rx 180 ry 0 rz 180 deg; joints [-68.351, 68.057, -90.27, 69.824, 98.017, 20.785]
  MoveL 10699 to (225.34, 164.63, 144.49) mm, rotated rx 180 ry 0 rz 180 deg; joints [-68.351, 68.057, -90.27, 69.824, 98.017, 20.785]
  Call Extruder(662.78032)
  MoveL 10700 to (225, 164.68, 144.49) mm, rotated rx -180 ry 0 rz -180 deg; joints [-68.461, 68.049, -90.274, 69.929, 97.982, 20.81]
  MoveL 10701 to (225, 164.68, 144.49) mm, rotated rx -180 ry 0 rz -180 deg; joints [-68.461, 68.049, -90.274, 69.929, 97.982, 20.81]
  Call Extruder(662.97876)
  MoveL 10702 to (224.61, 164.73, 144.49) mm, rotated rx 180 ry 0 rz 180 deg; joints [-68.583, 68.04, -90.277, 70.046, 97.943, 20.838]
  MoveL 10703 to (224.61, 164.73, 144.49) mm, rotated rx 180 ry 0 rz 180 deg; joints [-68.583, 68.04, -90.277, 70.046, 97.943, 20.838]
  Call Extruder(663.17634)
  MoveL 10704 to (224.22, 164.77, 144.49) mm, rotated rx 180 ry 0 rz 180 deg; joints [-68.706, 68.031, -90.281, 70.163, 97.904, 20.866]
  MoveL 10705 to (224.22, 164.77, 144.49) mm, rotated rx 180 ry 0 rz 180 deg; joints [-68.706, 68.031, -90.281, 70.163, 97.904, 20.866]
  Call Extruder(663.37305)
  MoveL 10706 to (223.83, 164.82, 144.49) mm, rotated rx 180 ry 0 rz 180 deg; joints [-68.828, 68.022, -90.285, 70.28, 97.864, 20.894]
  MoveL 10707 to (223.83, 164.82, 144.49) mm, rotated rx 180 ry 0 rz 180 deg; joints [-68.828, 68.022, -90.285, 70.28, 97.864, 20.894]
  Call Extruder(663.56888)
  MoveL 10708 to (223.45, 164.86, 144.49) mm, rotated rx 180 ry 0 rz -180 deg; joints [-68.951, 68.013, -90.289, 70.398, 97.825, 20.922]
  MoveL 10709 to (223.45, 164.86, 144.49) mm, rotated rx 180 ry 0 rz -180 deg; joints [-68.951, 68.013, -90.289, 70.398, 97.825, 20.922]
  Call Extruder(663.86424)
  MoveL 10710 to (222.86, 164.91, 144.49) mm, rotated rx 180 ry 0 rz 180 deg; joints [-69.135, 67.998, -90.296, 70.574, 97.767, 20.966]
  MoveL 10711 to (222.86, 164.91, 144.49) mm, rotated rx 180 ry 0 rz 180 deg; joints [-69.135, 67.998, -90.296, 70.574, 97.767, 20.966]
  Call Extruder(664.15827)
  MoveL 10712 to (222.27, 164.96, 144.49) mm, rotated rx 180 ry 0 rz 180 deg; joints [-69.319, 67.983, -90.302, 70.75, 97.708, 21.01]
  MoveL 10713 to (222.27, 164.96, 144.49) mm, rotated rx 180 ry 0 rz 180 deg; joints [-69.319, 67.983, -90.302, 70.75, 97.708, 21.01]
  Call Extruder(664.45096)
  MoveL 10714 to (221.68, 165, 144.49) mm, rotated rx 180 ry 0 rz 180 deg; joints [-69.504, 67.968, -90.309, 70.927, 97.649, 21.054]
  MoveL 10715 to (221.68, 165, 144.49) mm, rotated rx 180 ry 0 rz 180 deg; joints [-69.504, 67.968, -90.309, 70.927, 97.649, 21.054]
  Call Extruder(665.02441)
  MoveL 10716 to (220.52, 165.05, 144.49) mm, rotated rx -180 ry 0 rz -180 deg; joints [-69.864, 67.934, -90.323, 71.272, 97.534, 21.144]
  MoveL 10717 to (220.52, 165.05, 144.49) mm, rotated rx -180 ry 0 rz -180 deg; joints [-69.864, 67.934, -90.323, 71.272, 97.534, 21.144]
  Call Extruder(665.73842)
  MoveL 10718 to (219.06, 165.09, 144.49) mm, rotated rx 180 ry 0 rz 180 deg; joints [-70.315, 67.892, -90.341, 71.703, 97.39, 21.257]
  Call Extruder(782.58519)
  MoveL 10719 to (-19.06, 165.09, 144.49) mm, rotated rx -180 ry 0 rz 180 deg; joints [-137.325, 73.424, -86.804, 136.539, 80.204, 9.159]
  Call Extruder(783.01380)
  MoveL 10720 to (-19.94, 165.07, 144.49) mm, rotated rx -180 ry 0 rz -180 deg; joints [-137.467, 73.467, -86.763, 136.691, 80.243, 9.076]
  MoveL 10721 to (-19.94, 165.07, 144.49) mm, rotated rx -180 ry 0 rz -180 deg; joints [-137.467, 73.467, -86.763, 136.691, 80.243, 9.076]
  Call Extruder(783.58725)
  MoveL 10722 to (-21.1, 165.02, 144.49) mm, rotated rx 180 ry 0 rz -180 deg; joints [-137.659, 73.525, -86.709, 136.896, 80.294, 8.967]
  MoveL 10723 to (-21.1, 165.02, 144.49) mm, rotated rx 180 ry 0 rz -180 deg; joints [-137.659, 73.525, -86.709, 136.896, 80.294, 8.967]
  Call Extruder(784.02155)
  MoveL 10724 to (-21.97, 164.98, 144.49) mm, rotated rx 180 ry 0 rz 180 deg; joints [-137.804, 73.567, -86.669, 137.051, 80.332, 8.885]
  MoveL 10725 to (-21.97, 164.98, 144.49) mm, rotated rx 180 ry 0 rz 180 deg; joints [-137.804, 73.567, -86.669, 137.051, 80.332, 8.885]
  Call Extruder(784.31557)
  MoveL 10726 to (-22.56, 164.93, 144.49) mm, rotated rx 180 ry 0 rz 180 deg; joints [-137.905, 73.595, -86.642, 137.158, 80.356, 8.83]
  MoveL 10727 to (-22.56, 164.93, 144.49) mm, rotated rx 180 ry 0 rz 180 deg; joints [-137.905, 73.595, -86.642, 137.158, 80.356, 8.83]
  Call Extruder(784.61093)
  MoveL 10728 to (-23.15, 164.89, 144.49) mm, rotated rx 180 ry 0 rz -180 deg; joints [-138.004, 73.623, -86.616, 137.265, 80.381, 8.776]
  MoveL 10729 to (-23.15, 164.89, 144.49) mm, rotated rx 180 ry 0 rz -180 deg; joints [-138.004, 73.623, -86.616, 137.265, 80.381, 8.776]
  Call Extruder(784.85715)
  MoveL 10730 to (-23.64, 164.84, 144.49) mm, rotated rx 180 ry 0 rz 180 deg; joints [-138.088, 73.646, -86.594, 137.354, 80.401, 8.731]
  MoveL 10731 to (-23.64, 164.84, 144.49) mm, rotated rx 180 ry 0 rz 180 deg; joints [-138.088, 73.646, -86.594, 137.354, 80.401, 8.731]
  Call Extruder(785.05385)
  MoveL 10732 to (-24.03, 164.79, 144.49) mm, rotated rx -180 ry 0 rz 180 deg; joints [-138.156, 73.663, -86.577, 137.426, 80.416, 8.696]
  MoveL 10733 to (-24.03, 164.79, 144.49) mm, rotated rx -180 ry 0 rz 180 deg; joints [-138.156, 73.663, -86.577, 137.426, 80.416, 8.696]
  Call Extruder(785.25143)
  MoveL 10734 to (-24.42, 164.75, 144.49) mm, rotated rx 180 ry 0 rz 180 deg; joints [-138.224, 73.681, -86.56, 137.498, 80.432, 8.661]
  MoveL 10735 to (-24.42, 164.75, 144.49) mm, rotated rx 180 ry 0 rz 180 deg; joints [-138.224, 73.681, -86.56, 137.498, 80.432, 8.661]
  Call Extruder(785.44987)
  MoveL 10736 to (-24.8, 164.7, 144.49) mm, rotated rx -180 ry 0 rz 180 deg; joints [-138.292, 73.698, -86.543, 137.57, 80.447, 8.626]
  MoveL 10737 to (-24.8, 164.7, 144.49) mm, rotated rx -180 ry 0 rz 180 deg; joints [-138.292, 73.698, -86.543, 137.57, 80.447, 8.626]
  Call Extruder(785.64918)
  MoveL 10738 to (-25.19, 164.66, 144.49) mm, rotated rx -180 ry 0 rz 180 deg; joints [-138.359, 73.716, -86.526, 137.641, 80.463, 8.591]
  MoveL 10739 to (-25.19, 164.66, 144.49) mm, rotated rx -180 ry 0 rz 180 deg; joints [-138.359, 73.716, -86.526, 137.641, 80.463, 8.591]
  Call Extruder(785.80801)
  MoveL 10740 to (-25.5, 164.61, 144.49) mm, rotated rx 180 ry 0 rz -180 deg; joints [-138.415, 73.729, -86.512, 137.7, 80.474, 8.564]
  MoveL 10741 to (-25.5, 164.61, 144.49) mm, rotated rx 180 ry 0 rz -180 deg; joints [-138.415, 73.729, -86.512, 137.7, 80.474, 8.564]
  Call Extruder(785.96757)
  MoveL 10742 to (-25.8, 164.56, 144.49) mm, rotated rx -180 ry 0 rz -180 deg; joints [-138.47, 73.743, -86.499, 137.758, 80.485, 8.537]
  MoveL 10743 to (-25.8, 164.56, 144.49) mm, rotated rx -180 ry 0 rz -180 deg; joints [-138.47, 73.743, -86.499, 137.758, 80.485, 8.537]
  Call Extruder(786.12786)
  MoveL 10744 to (-26.11, 164.51, 144.49) mm, rotated rx -180 ry 0 rz 180 deg; joints [-138.525, 73.756, -86.486, 137.816, 80.497, 8.51]
  MoveL 10745 to (-26.11, 164.51, 144.49) mm, rotated rx -180 ry 0 rz 180 deg; joints [-138.525, 73.756, -86.486, 137.816, 80.497, 8.51]
  Call Extruder(786.28887)
